REGION Network 54: Reset CMS
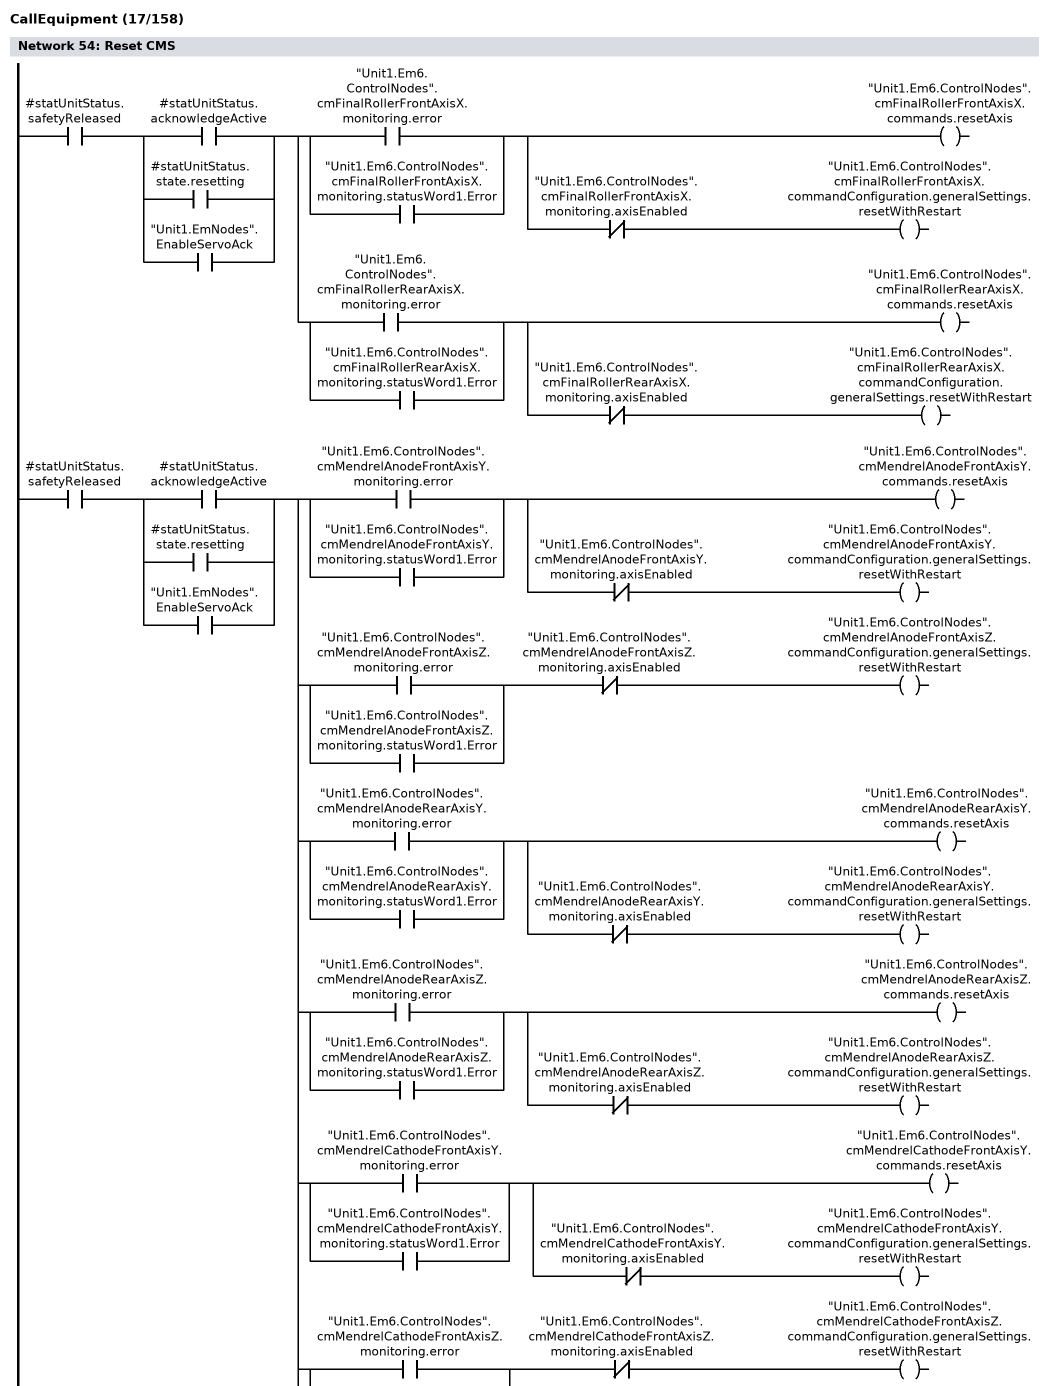
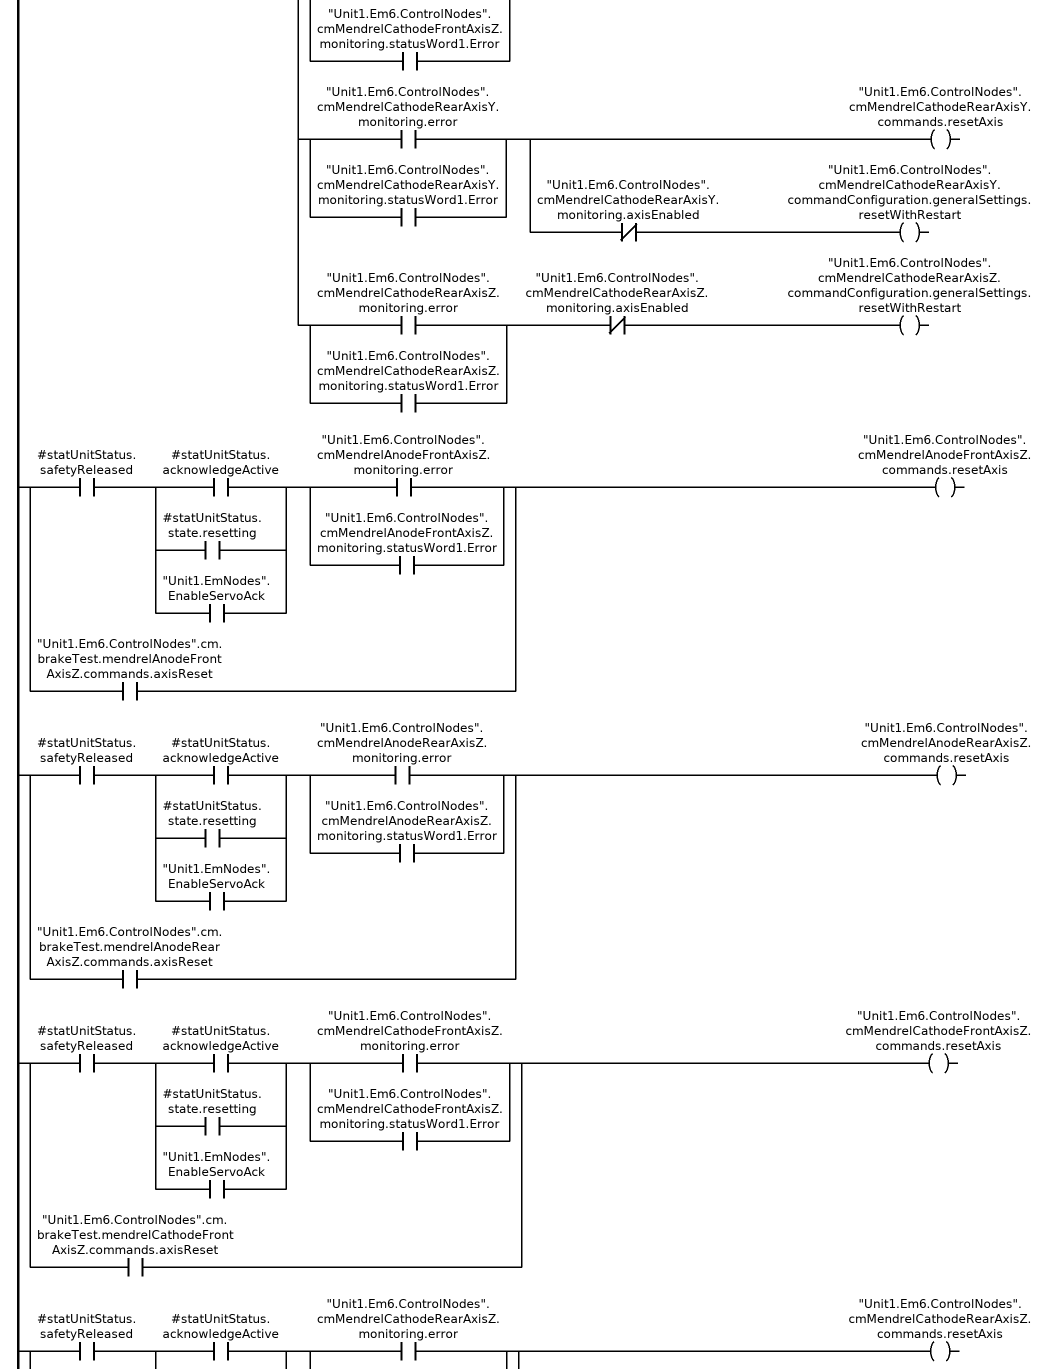
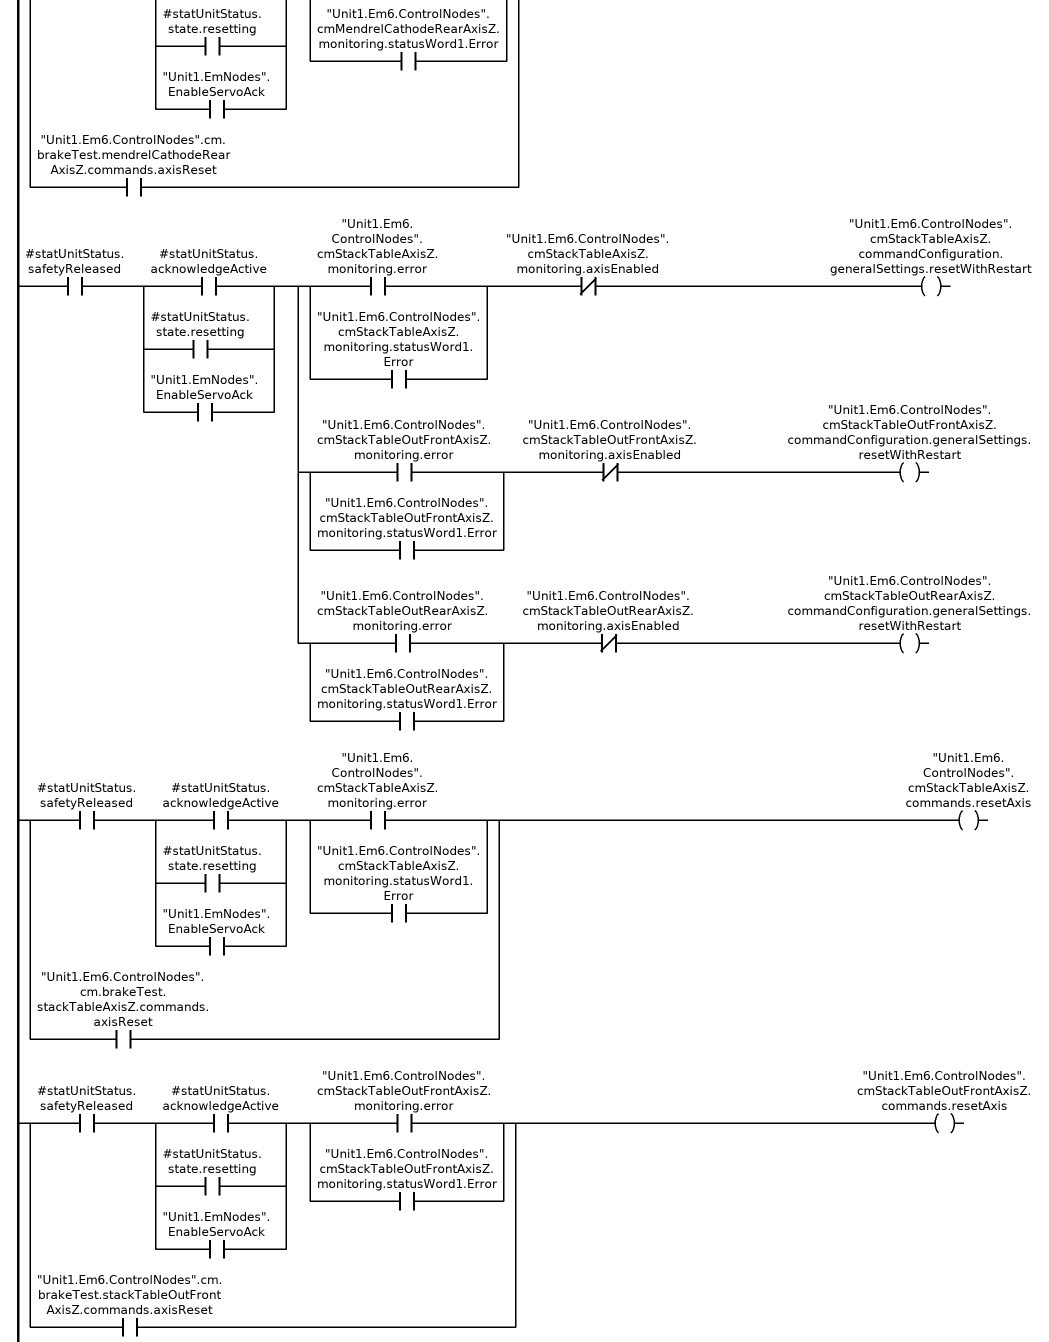
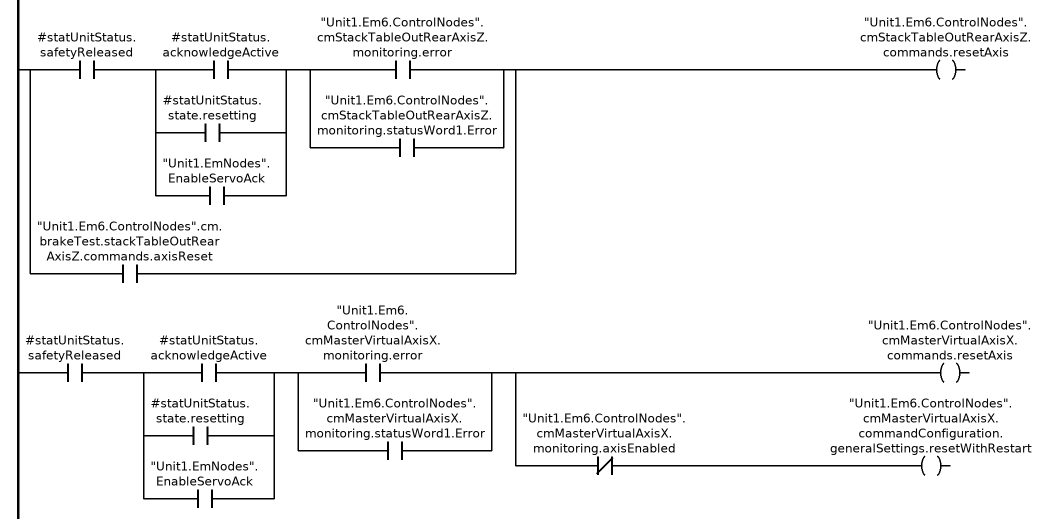
   RUNG wire#powerrail
      Contact( #statUnitStatus.safetyReleased )
      wire#w1
      Contact( #statUnitStatus.acknowledgeActive )
      wire#w2
      Contact( "Unit1.Em6.ControlNodes".cmFinalRollerFrontAxisX.monitoring.error )
      wire#w3
      Coil( "Unit1.Em6.ControlNodes".cmFinalRollerFrontAxisX.commands.resetAxis )
   END_RUNG
   RUNG wire#w1
      Contact( #statUnitStatus.state.resetting )
   END_RUNG wire#w2
   RUNG wire#w1
      Contact( "Unit1.EmNodes".EnableServoAck )
   END_RUNG wire#w2
   RUNG wire#w2
      Contact( "Unit1.Em6.ControlNodes".cmFinalRollerFrontAxisX.monitoring.statusWord1.Error )
   END_RUNG wire#w3
   RUNG wire#w3
      I_Contact( "Unit1.Em6.ControlNodes".cmFinalRollerFrontAxisX.monitoring.axisEnabled )
      Coil( "Unit1.Em6.ControlNodes".cmFinalRollerFrontAxisX.commandConfiguration.generalSettings.resetWithRestart )
   END_RUNG
   RUNG wire#w2
      Contact( "Unit1.Em6.ControlNodes".cmFinalRollerRearAxisX.monitoring.error )
      wire#w4
      Coil( "Unit1.Em6.ControlNodes".cmFinalRollerRearAxisX.commands.resetAxis )
   END_RUNG
   RUNG wire#w2
      Contact( "Unit1.Em6.ControlNodes".cmFinalRollerRearAxisX.monitoring.statusWord1.Error )
   END_RUNG wire#w4
   RUNG wire#w4
      I_Contact( "Unit1.Em6.ControlNodes".cmFinalRollerRearAxisX.monitoring.axisEnabled )
      Coil( "Unit1.Em6.ControlNodes".cmFinalRollerRearAxisX.commandConfiguration.generalSettings.resetWithRestart )
   END_RUNG
   RUNG wire#powerrail
      Contact( #statUnitStatus.safetyReleased )
      wire#w5
      Contact( #statUnitStatus.acknowledgeActive )
      wire#w6
      Contact( "Unit1.Em6.ControlNodes".cmMendrelAnodeFrontAxisY.monitoring.error )
      wire#w7
      Coil( "Unit1.Em6.ControlNodes".cmMendrelAnodeFrontAxisY.commands.resetAxis )
   END_RUNG
   RUNG wire#w5
      Contact( #statUnitStatus.state.resetting )
   END_RUNG wire#w6
   RUNG wire#w5
      Contact( "Unit1.EmNodes".EnableServoAck )
   END_RUNG wire#w6
   RUNG wire#w6
      Contact( "Unit1.Em6.ControlNodes".cmMendrelAnodeFrontAxisY.monitoring.statusWord1.Error )
   END_RUNG wire#w7
   RUNG wire#w7
      I_Contact( "Unit1.Em6.ControlNodes".cmMendrelAnodeFrontAxisY.monitoring.axisEnabled )
      Coil( "Unit1.Em6.ControlNodes".cmMendrelAnodeFrontAxisY.commandConfiguration.generalSettings.resetWithRestart )
   END_RUNG
   RUNG wire#w6
      Contact( "Unit1.Em6.ControlNodes".cmMendrelAnodeFrontAxisZ.monitoring.error )
      wire#w8
      I_Contact( "Unit1.Em6.ControlNodes".cmMendrelAnodeFrontAxisZ.monitoring.axisEnabled )
      Coil( "Unit1.Em6.ControlNodes".cmMendrelAnodeFrontAxisZ.commandConfiguration.generalSettings.resetWithRestart )
   END_RUNG
   RUNG wire#w6
      Contact( "Unit1.Em6.ControlNodes".cmMendrelAnodeFrontAxisZ.monitoring.statusWord1.Error )
   END_RUNG wire#w8
   RUNG wire#w6
      Contact( "Unit1.Em6.ControlNodes".cmMendrelAnodeRearAxisY.monitoring.error )
      wire#w9
      Coil( "Unit1.Em6.ControlNodes".cmMendrelAnodeRearAxisY.commands.resetAxis )
   END_RUNG
   RUNG wire#w6
      Contact( "Unit1.Em6.ControlNodes".cmMendrelAnodeRearAxisY.monitoring.statusWord1.Error )
   END_RUNG wire#w9
   RUNG wire#w9
      I_Contact( "Unit1.Em6.ControlNodes".cmMendrelAnodeRearAxisY.monitoring.axisEnabled )
      Coil( "Unit1.Em6.ControlNodes".cmMendrelAnodeRearAxisY.commandConfiguration.generalSettings.resetWithRestart )
   END_RUNG
   RUNG wire#w6
      Contact( "Unit1.Em6.ControlNodes".cmMendrelAnodeRearAxisZ.monitoring.error )
      wire#w10
      Coil( "Unit1.Em6.ControlNodes".cmMendrelAnodeRearAxisZ.commands.resetAxis )
   END_RUNG
   RUNG wire#w6
      Contact( "Unit1.Em6.ControlNodes".cmMendrelAnodeRearAxisZ.monitoring.statusWord1.Error )
   END_RUNG wire#w10
   RUNG wire#w10
      I_Contact( "Unit1.Em6.ControlNodes".cmMendrelAnodeRearAxisZ.monitoring.axisEnabled )
      Coil( "Unit1.Em6.ControlNodes".cmMendrelAnodeRearAxisZ.commandConfiguration.generalSettings.resetWithRestart )
   END_RUNG
   RUNG wire#w6
      Contact( "Unit1.Em6.ControlNodes".cmMendrelCathodeFrontAxisY.monitoring.error )
      wire#w11
      Coil( "Unit1.Em6.ControlNodes".cmMendrelCathodeFrontAxisY.commands.resetAxis )
   END_RUNG
   RUNG wire#w6
      Contact( "Unit1.Em6.ControlNodes".cmMendrelCathodeFrontAxisY.monitoring.statusWord1.Error )
   END_RUNG wire#w11
   RUNG wire#w11
      I_Contact( "Unit1.Em6.ControlNodes".cmMendrelCathodeFrontAxisY.monitoring.axisEnabled )
      Coil( "Unit1.Em6.ControlNodes".cmMendrelCathodeFrontAxisY.commandConfiguration.generalSettings.resetWithRestart )
   END_RUNG
   RUNG wire#w6
      Contact( "Unit1.Em6.ControlNodes".cmMendrelCathodeFrontAxisZ.monitoring.error )
      wire#w12
      I_Contact( "Unit1.Em6.ControlNodes".cmMendrelCathodeFrontAxisZ.monitoring.axisEnabled )
      Coil( "Unit1.Em6.ControlNodes".cmMendrelCathodeFrontAxisZ.commandConfiguration.generalSettings.resetWithRestart )
   END_RUNG
   RUNG wire#w6
      Contact( "Unit1.Em6.ControlNodes".cmMendrelCathodeFrontAxisZ.monitoring.statusWord1.Error )
   END_RUNG wire#w12
   RUNG wire#w6
      Contact( "Unit1.Em6.ControlNodes".cmMendrelCathodeRearAxisY.monitoring.error )
      wire#w13
      Coil( "Unit1.Em6.ControlNodes".cmMendrelCathodeRearAxisY.commands.resetAxis )
   END_RUNG
   RUNG wire#w6
      Contact( "Unit1.Em6.ControlNodes".cmMendrelCathodeRearAxisY.monitoring.statusWord1.Error )
   END_RUNG wire#w13
   RUNG wire#w13
      I_Contact( "Unit1.Em6.ControlNodes".cmMendrelCathodeRearAxisY.monitoring.axisEnabled )
      Coil( "Unit1.Em6.ControlNodes".cmMendrelCathodeRearAxisY.commandConfiguration.generalSettings.resetWithRestart )
   END_RUNG
   RUNG wire#w6
      Contact( "Unit1.Em6.ControlNodes".cmMendrelCathodeRearAxisZ.monitoring.error )
      wire#w14
      I_Contact( "Unit1.Em6.ControlNodes".cmMendrelCathodeRearAxisZ.monitoring.axisEnabled )
      Coil( "Unit1.Em6.ControlNodes".cmMendrelCathodeRearAxisZ.commandConfiguration.generalSettings.resetWithRestart )
   END_RUNG
   RUNG wire#w6
      Contact( "Unit1.Em6.ControlNodes".cmMendrelCathodeRearAxisZ.monitoring.statusWord1.Error )
   END_RUNG wire#w14
   RUNG wire#powerrail
      Contact( #statUnitStatus.safetyReleased )
      wire#w15
      Contact( #statUnitStatus.acknowledgeActive )
      wire#w16
      Contact( "Unit1.Em6.ControlNodes".cmMendrelAnodeFrontAxisZ.monitoring.error )
      wire#w17
      Coil( "Unit1.Em6.ControlNodes".cmMendrelAnodeFrontAxisZ.commands.resetAxis )
   END_RUNG
   RUNG wire#w15
      Contact( #statUnitStatus.state.resetting )
   END_RUNG wire#w16
   RUNG wire#w15
      Contact( "Unit1.EmNodes".EnableServoAck )
   END_RUNG wire#w16
   RUNG wire#w16
      Contact( "Unit1.Em6.ControlNodes".cmMendrelAnodeFrontAxisZ.monitoring.statusWord1.Error )
   END_RUNG wire#w17
   RUNG wire#powerrail
      Contact( "Unit1.Em6.ControlNodes".cm.brakeTest.mendrelAnodeFrontAxisZ.commands.axisReset )
   END_RUNG wire#w17
   RUNG wire#powerrail
      Contact( #statUnitStatus.safetyReleased )
      wire#w18
      Contact( #statUnitStatus.acknowledgeActive )
      wire#w19
      Contact( "Unit1.Em6.ControlNodes".cmMendrelAnodeRearAxisZ.monitoring.error )
      wire#w20
      Coil( "Unit1.Em6.ControlNodes".cmMendrelAnodeRearAxisZ.commands.resetAxis )
   END_RUNG
   RUNG wire#w18
      Contact( #statUnitStatus.state.resetting )
   END_RUNG wire#w19
   RUNG wire#w18
      Contact( "Unit1.EmNodes".EnableServoAck )
   END_RUNG wire#w19
   RUNG wire#w19
      Contact( "Unit1.Em6.ControlNodes".cmMendrelAnodeRearAxisZ.monitoring.statusWord1.Error )
   END_RUNG wire#w20
   RUNG wire#powerrail
      Contact( "Unit1.Em6.ControlNodes".cm.brakeTest.mendrelAnodeRearAxisZ.commands.axisReset )
   END_RUNG wire#w20
   RUNG wire#powerrail
      Contact( #statUnitStatus.safetyReleased )
      wire#w21
      Contact( #statUnitStatus.acknowledgeActive )
      wire#w22
      Contact( "Unit1.Em6.ControlNodes".cmMendrelCathodeFrontAxisZ.monitoring.error )
      wire#w23
      Coil( "Unit1.Em6.ControlNodes".cmMendrelCathodeFrontAxisZ.commands.resetAxis )
   END_RUNG
   RUNG wire#w21
      Contact( #statUnitStatus.state.resetting )
   END_RUNG wire#w22
   RUNG wire#w21
      Contact( "Unit1.EmNodes".EnableServoAck )
   END_RUNG wire#w22
   RUNG wire#w22
      Contact( "Unit1.Em6.ControlNodes".cmMendrelCathodeFrontAxisZ.monitoring.statusWord1.Error )
   END_RUNG wire#w23
   RUNG wire#powerrail
      Contact( "Unit1.Em6.ControlNodes".cm.brakeTest.mendrelCathodeFrontAxisZ.commands.axisReset )
   END_RUNG wire#w23
   RUNG wire#powerrail
      Contact( #statUnitStatus.safetyReleased )
      wire#w24
      Contact( #statUnitStatus.acknowledgeActive )
      wire#w25
      Contact( "Unit1.Em6.ControlNodes".cmMendrelCathodeRearAxisZ.monitoring.error )
      wire#w26
      Coil( "Unit1.Em6.ControlNodes".cmMendrelCathodeRearAxisZ.commands.resetAxis )
   END_RUNG
   RUNG wire#w24
      Contact( #statUnitStatus.state.resetting )
   END_RUNG wire#w25
   RUNG wire#w24
      Contact( "Unit1.EmNodes".EnableServoAck )
   END_RUNG wire#w25
   RUNG wire#w25
      Contact( "Unit1.Em6.ControlNodes".cmMendrelCathodeRearAxisZ.monitoring.statusWord1.Error )
   END_RUNG wire#w26
   RUNG wire#powerrail
      Contact( "Unit1.Em6.ControlNodes".cm.brakeTest.mendrelCathodeRearAxisZ.commands.axisReset )
   END_RUNG wire#w26
   RUNG wire#powerrail
      Contact( #statUnitStatus.safetyReleased )
      wire#w27
      Contact( #statUnitStatus.acknowledgeActive )
      wire#w28
      Contact( "Unit1.Em6.ControlNodes".cmStackTableAxisZ.monitoring.error )
      wire#w29
      I_Contact( "Unit1.Em6.ControlNodes".cmStackTableAxisZ.monitoring.axisEnabled )
      Coil( "Unit1.Em6.ControlNodes".cmStackTableAxisZ.commandConfiguration.generalSettings.resetWithRestart )
   END_RUNG
   RUNG wire#w27
      Contact( #statUnitStatus.state.resetting )
   END_RUNG wire#w28
   RUNG wire#w27
      Contact( "Unit1.EmNodes".EnableServoAck )
   END_RUNG wire#w28
   RUNG wire#w28
      Contact( "Unit1.Em6.ControlNodes".cmStackTableAxisZ.monitoring.statusWord1.Error )
   END_RUNG wire#w29
   RUNG wire#w28
      Contact( "Unit1.Em6.ControlNodes".cmStackTableOutFrontAxisZ.monitoring.error )
      wire#w30
      I_Contact( "Unit1.Em6.ControlNodes".cmStackTableOutFrontAxisZ.monitoring.axisEnabled )
      Coil( "Unit1.Em6.ControlNodes".cmStackTableOutFrontAxisZ.commandConfiguration.generalSettings.resetWithRestart )
   END_RUNG
   RUNG wire#w28
      Contact( "Unit1.Em6.ControlNodes".cmStackTableOutFrontAxisZ.monitoring.statusWord1.Error )
   END_RUNG wire#w30
   RUNG wire#w28
      Contact( "Unit1.Em6.ControlNodes".cmStackTableOutRearAxisZ.monitoring.error )
      wire#w31
      I_Contact( "Unit1.Em6.ControlNodes".cmStackTableOutRearAxisZ.monitoring.axisEnabled )
      Coil( "Unit1.Em6.ControlNodes".cmStackTableOutRearAxisZ.commandConfiguration.generalSettings.resetWithRestart )
   END_RUNG
   RUNG wire#w28
      Contact( "Unit1.Em6.ControlNodes".cmStackTableOutRearAxisZ.monitoring.statusWord1.Error )
   END_RUNG wire#w31
   RUNG wire#powerrail
      Contact( #statUnitStatus.safetyReleased )
      wire#w32
      Contact( #statUnitStatus.acknowledgeActive )
      wire#w33
      Contact( "Unit1.Em6.ControlNodes".cmStackTableAxisZ.monitoring.error )
      wire#w34
      Coil( "Unit1.Em6.ControlNodes".cmStackTableAxisZ.commands.resetAxis )
   END_RUNG
   RUNG wire#w32
      Contact( #statUnitStatus.state.resetting )
   END_RUNG wire#w33
   RUNG wire#w32
      Contact( "Unit1.EmNodes".EnableServoAck )
   END_RUNG wire#w33
   RUNG wire#w33
      Contact( "Unit1.Em6.ControlNodes".cmStackTableAxisZ.monitoring.statusWord1.Error )
   END_RUNG wire#w34
   RUNG wire#powerrail
      Contact( "Unit1.Em6.ControlNodes".cm.brakeTest.stackTableAxisZ.commands.axisReset )
   END_RUNG wire#w34
   RUNG wire#powerrail
      Contact( #statUnitStatus.safetyReleased )
      wire#w35
      Contact( #statUnitStatus.acknowledgeActive )
      wire#w36
      Contact( "Unit1.Em6.ControlNodes".cmStackTableOutFrontAxisZ.monitoring.error )
      wire#w37
      Coil( "Unit1.Em6.ControlNodes".cmStackTableOutFrontAxisZ.commands.resetAxis )
   END_RUNG
   RUNG wire#w35
      Contact( #statUnitStatus.state.resetting )
   END_RUNG wire#w36
   RUNG wire#w35
      Contact( "Unit1.EmNodes".EnableServoAck )
   END_RUNG wire#w36
   RUNG wire#w36
      Contact( "Unit1.Em6.ControlNodes".cmStackTableOutFrontAxisZ.monitoring.statusWord1.Error )
   END_RUNG wire#w37
   RUNG wire#powerrail
      Contact( "Unit1.Em6.ControlNodes".cm.brakeTest.stackTableOutFrontAxisZ.commands.axisReset )
   END_RUNG wire#w37
   RUNG wire#powerrail
      Contact( #statUnitStatus.safetyReleased )
      wire#w38
      Contact( #statUnitStatus.acknowledgeActive )
      wire#w39
      Contact( "Unit1.Em6.ControlNodes".cmStackTableOutRearAxisZ.monitoring.error )
      wire#w40
      Coil( "Unit1.Em6.ControlNodes".cmStackTableOutRearAxisZ.commands.resetAxis )
   END_RUNG
   RUNG wire#w38
      Contact( #statUnitStatus.state.resetting )
   END_RUNG wire#w39
   RUNG wire#w38
      Contact( "Unit1.EmNodes".EnableServoAck )
   END_RUNG wire#w39
   RUNG wire#w39
      Contact( "Unit1.Em6.ControlNodes".cmStackTableOutRearAxisZ.monitoring.statusWord1.Error )
   END_RUNG wire#w40
   RUNG wire#powerrail
      Contact( "Unit1.Em6.ControlNodes".cm.brakeTest.stackTableOutRearAxisZ.commands.axisReset )
   END_RUNG wire#w40
   RUNG wire#powerrail
      Contact( #statUnitStatus.safetyReleased )
      wire#w41
      Contact( #statUnitStatus.acknowledgeActive )
      wire#w42
      Contact( "Unit1.Em6.ControlNodes".cmMasterVirtualAxisX.monitoring.error )
      wire#w43
      Coil( "Unit1.Em6.ControlNodes".cmMasterVirtualAxisX.commands.resetAxis )
   END_RUNG
   RUNG wire#w41
      Contact( #statUnitStatus.state.resetting )
   END_RUNG wire#w42
   RUNG wire#w41
      Contact( "Unit1.EmNodes".EnableServoAck )
   END_RUNG wire#w42
   RUNG wire#w42
      Contact( "Unit1.Em6.ControlNodes".cmMasterVirtualAxisX.monitoring.statusWord1.Error )
   END_RUNG wire#w43
   RUNG wire#w43
      I_Contact( "Unit1.Em6.ControlNodes".cmMasterVirtualAxisX.monitoring.axisEnabled )
      Coil( "Unit1.Em6.ControlNodes".cmMasterVirtualAxisX.commandConfiguration.generalSettings.resetWithRestart )
   END_RUNG
   // the same network as SCL:
   #_w1 := #statUnitStatus.safetyReleased AND (#statUnitStatus.acknowledgeActive OR #statUnitStatus.state.resetting OR "Unit1.EmNodes".EnableServoAck);
   "Unit1.Em6.ControlNodes".cmFinalRollerFrontAxisX.commands.resetAxis := #_w1 AND ("Unit1.Em6.ControlNodes".cmFinalRollerFrontAxisX.monitoring.error OR "Unit1.Em6.ControlNodes".cmFinalRollerFrontAxisX.monitoring.statusWord1.Error);
   "Unit1.Em6.ControlNodes".cmFinalRollerFrontAxisX.commandConfiguration.generalSettings.resetWithRestart := "Unit1.Em6.ControlNodes".cmFinalRollerFrontAxisX.commands.resetAxis AND NOT "Unit1.Em6.ControlNodes".cmFinalRollerFrontAxisX.monitoring.axisEnabled;
   "Unit1.Em6.ControlNodes".cmFinalRollerRearAxisX.commands.resetAxis := #_w1 AND ("Unit1.Em6.ControlNodes".cmFinalRollerRearAxisX.monitoring.error OR "Unit1.Em6.ControlNodes".cmFinalRollerRearAxisX.monitoring.statusWord1.Error);
   "Unit1.Em6.ControlNodes".cmFinalRollerRearAxisX.commandConfiguration.generalSettings.resetWithRestart := "Unit1.Em6.ControlNodes".cmFinalRollerRearAxisX.commands.resetAxis AND NOT "Unit1.Em6.ControlNodes".cmFinalRollerRearAxisX.monitoring.axisEnabled;
   #_w2 := #statUnitStatus.safetyReleased AND (#statUnitStatus.acknowledgeActive OR #statUnitStatus.state.resetting OR "Unit1.EmNodes".EnableServoAck);
   "Unit1.Em6.ControlNodes".cmMendrelAnodeFrontAxisY.commands.resetAxis := #_w2 AND ("Unit1.Em6.ControlNodes".cmMendrelAnodeFrontAxisY.monitoring.error OR "Unit1.Em6.ControlNodes".cmMendrelAnodeFrontAxisY.monitoring.statusWord1.Error);
   "Unit1.Em6.ControlNodes".cmMendrelAnodeFrontAxisY.commandConfiguration.generalSettings.resetWithRestart := "Unit1.Em6.ControlNodes".cmMendrelAnodeFrontAxisY.commands.resetAxis AND NOT "Unit1.Em6.ControlNodes".cmMendrelAnodeFrontAxisY.monitoring.axisEnabled;
   "Unit1.Em6.ControlNodes".cmMendrelAnodeFrontAxisZ.commandConfiguration.generalSettings.resetWithRestart := #_w2 AND ("Unit1.Em6.ControlNodes".cmMendrelAnodeFrontAxisZ.monitoring.error OR "Unit1.Em6.ControlNodes".cmMendrelAnodeFrontAxisZ.monitoring.statusWord1.Error) AND NOT "Unit1.Em6.ControlNodes".cmMendrelAnodeFrontAxisZ.monitoring.axisEnabled;
   "Unit1.Em6.ControlNodes".cmMendrelAnodeRearAxisY.commands.resetAxis := #_w2 AND ("Unit1.Em6.ControlNodes".cmMendrelAnodeRearAxisY.monitoring.error OR "Unit1.Em6.ControlNodes".cmMendrelAnodeRearAxisY.monitoring.statusWord1.Error);
   "Unit1.Em6.ControlNodes".cmMendrelAnodeRearAxisY.commandConfiguration.generalSettings.resetWithRestart := "Unit1.Em6.ControlNodes".cmMendrelAnodeRearAxisY.commands.resetAxis AND NOT "Unit1.Em6.ControlNodes".cmMendrelAnodeRearAxisY.monitoring.axisEnabled;
   "Unit1.Em6.ControlNodes".cmMendrelAnodeRearAxisZ.commands.resetAxis := #_w2 AND ("Unit1.Em6.ControlNodes".cmMendrelAnodeRearAxisZ.monitoring.error OR "Unit1.Em6.ControlNodes".cmMendrelAnodeRearAxisZ.monitoring.statusWord1.Error);
   "Unit1.Em6.ControlNodes".cmMendrelAnodeRearAxisZ.commandConfiguration.generalSettings.resetWithRestart := "Unit1.Em6.ControlNodes".cmMendrelAnodeRearAxisZ.commands.resetAxis AND NOT "Unit1.Em6.ControlNodes".cmMendrelAnodeRearAxisZ.monitoring.axisEnabled;
   "Unit1.Em6.ControlNodes".cmMendrelCathodeFrontAxisY.commands.resetAxis := #_w2 AND ("Unit1.Em6.ControlNodes".cmMendrelCathodeFrontAxisY.monitoring.error OR "Unit1.Em6.ControlNodes".cmMendrelCathodeFrontAxisY.monitoring.statusWord1.Error);
   "Unit1.Em6.ControlNodes".cmMendrelCathodeFrontAxisY.commandConfiguration.generalSettings.resetWithRestart := "Unit1.Em6.ControlNodes".cmMendrelCathodeFrontAxisY.commands.resetAxis AND NOT "Unit1.Em6.ControlNodes".cmMendrelCathodeFrontAxisY.monitoring.axisEnabled;
   "Unit1.Em6.ControlNodes".cmMendrelCathodeFrontAxisZ.commandConfiguration.generalSettings.resetWithRestart := #_w2 AND ("Unit1.Em6.ControlNodes".cmMendrelCathodeFrontAxisZ.monitoring.error OR "Unit1.Em6.ControlNodes".cmMendrelCathodeFrontAxisZ.monitoring.statusWord1.Error) AND NOT "Unit1.Em6.ControlNodes".cmMendrelCathodeFrontAxisZ.monitoring.axisEnabled;
   "Unit1.Em6.ControlNodes".cmMendrelCathodeRearAxisY.commands.resetAxis := #_w2 AND ("Unit1.Em6.ControlNodes".cmMendrelCathodeRearAxisY.monitoring.error OR "Unit1.Em6.ControlNodes".cmMendrelCathodeRearAxisY.monitoring.statusWord1.Error);
   "Unit1.Em6.ControlNodes".cmMendrelCathodeRearAxisY.commandConfiguration.generalSettings.resetWithRestart := "Unit1.Em6.ControlNodes".cmMendrelCathodeRearAxisY.commands.resetAxis AND NOT "Unit1.Em6.ControlNodes".cmMendrelCathodeRearAxisY.monitoring.axisEnabled;
   "Unit1.Em6.ControlNodes".cmMendrelCathodeRearAxisZ.commandConfiguration.generalSettings.resetWithRestart := #_w2 AND ("Unit1.Em6.ControlNodes".cmMendrelCathodeRearAxisZ.monitoring.error OR "Unit1.Em6.ControlNodes".cmMendrelCathodeRearAxisZ.monitoring.statusWord1.Error) AND NOT "Unit1.Em6.ControlNodes".cmMendrelCathodeRearAxisZ.monitoring.axisEnabled;
   "Unit1.Em6.ControlNodes".cmMendrelAnodeFrontAxisZ.commands.resetAxis := (#statUnitStatus.safetyReleased AND (#statUnitStatus.acknowledgeActive OR #statUnitStatus.state.resetting OR "Unit1.EmNodes".EnableServoAck) AND ("Unit1.Em6.ControlNodes".cmMendrelAnodeFrontAxisZ.monitoring.error OR "Unit1.Em6.ControlNodes".cmMendrelAnodeFrontAxisZ.monitoring.statusWord1.Error)) OR "Unit1.Em6.ControlNodes".cm.brakeTest.mendrelAnodeFrontAxisZ.commands.axisReset;
   "Unit1.Em6.ControlNodes".cmMendrelAnodeRearAxisZ.commands.resetAxis := (#statUnitStatus.safetyReleased AND (#statUnitStatus.acknowledgeActive OR #statUnitStatus.state.resetting OR "Unit1.EmNodes".EnableServoAck) AND ("Unit1.Em6.ControlNodes".cmMendrelAnodeRearAxisZ.monitoring.error OR "Unit1.Em6.ControlNodes".cmMendrelAnodeRearAxisZ.monitoring.statusWord1.Error)) OR "Unit1.Em6.ControlNodes".cm.brakeTest.mendrelAnodeRearAxisZ.commands.axisReset;
   "Unit1.Em6.ControlNodes".cmMendrelCathodeFrontAxisZ.commands.resetAxis := (#statUnitStatus.safetyReleased AND (#statUnitStatus.acknowledgeActive OR #statUnitStatus.state.resetting OR "Unit1.EmNodes".EnableServoAck) AND ("Unit1.Em6.ControlNodes".cmMendrelCathodeFrontAxisZ.monitoring.error OR "Unit1.Em6.ControlNodes".cmMendrelCathodeFrontAxisZ.monitoring.statusWord1.Error)) OR "Unit1.Em6.ControlNodes".cm.brakeTest.mendrelCathodeFrontAxisZ.commands.axisReset;
   "Unit1.Em6.ControlNodes".cmMendrelCathodeRearAxisZ.commands.resetAxis := (#statUnitStatus.safetyReleased AND (#statUnitStatus.acknowledgeActive OR #statUnitStatus.state.resetting OR "Unit1.EmNodes".EnableServoAck) AND ("Unit1.Em6.ControlNodes".cmMendrelCathodeRearAxisZ.monitoring.error OR "Unit1.Em6.ControlNodes".cmMendrelCathodeRearAxisZ.monitoring.statusWord1.Error)) OR "Unit1.Em6.ControlNodes".cm.brakeTest.mendrelCathodeRearAxisZ.commands.axisReset;
   #_w3 := #statUnitStatus.safetyReleased AND (#statUnitStatus.acknowledgeActive OR #statUnitStatus.state.resetting OR "Unit1.EmNodes".EnableServoAck);
   "Unit1.Em6.ControlNodes".cmStackTableAxisZ.commandConfiguration.generalSettings.resetWithRestart := #_w3 AND ("Unit1.Em6.ControlNodes".cmStackTableAxisZ.monitoring.error OR "Unit1.Em6.ControlNodes".cmStackTableAxisZ.monitoring.statusWord1.Error) AND NOT "Unit1.Em6.ControlNodes".cmStackTableAxisZ.monitoring.axisEnabled;
   "Unit1.Em6.ControlNodes".cmStackTableOutFrontAxisZ.commandConfiguration.generalSettings.resetWithRestart := #_w3 AND ("Unit1.Em6.ControlNodes".cmStackTableOutFrontAxisZ.monitoring.error OR "Unit1.Em6.ControlNodes".cmStackTableOutFrontAxisZ.monitoring.statusWord1.Error) AND NOT "Unit1.Em6.ControlNodes".cmStackTableOutFrontAxisZ.monitoring.axisEnabled;
   "Unit1.Em6.ControlNodes".cmStackTableOutRearAxisZ.commandConfiguration.generalSettings.resetWithRestart := #_w3 AND ("Unit1.Em6.ControlNodes".cmStackTableOutRearAxisZ.monitoring.error OR "Unit1.Em6.ControlNodes".cmStackTableOutRearAxisZ.monitoring.statusWord1.Error) AND NOT "Unit1.Em6.ControlNodes".cmStackTableOutRearAxisZ.monitoring.axisEnabled;
   "Unit1.Em6.ControlNodes".cmStackTableAxisZ.commands.resetAxis := (#statUnitStatus.safetyReleased AND (#statUnitStatus.acknowledgeActive OR #statUnitStatus.state.resetting OR "Unit1.EmNodes".EnableServoAck) AND ("Unit1.Em6.ControlNodes".cmStackTableAxisZ.monitoring.error OR "Unit1.Em6.ControlNodes".cmStackTableAxisZ.monitoring.statusWord1.Error)) OR "Unit1.Em6.ControlNodes".cm.brakeTest.stackTableAxisZ.commands.axisReset;
   "Unit1.Em6.ControlNodes".cmStackTableOutFrontAxisZ.commands.resetAxis := (#statUnitStatus.safetyReleased AND (#statUnitStatus.acknowledgeActive OR #statUnitStatus.state.resetting OR "Unit1.EmNodes".EnableServoAck) AND ("Unit1.Em6.ControlNodes".cmStackTableOutFrontAxisZ.monitoring.error OR "Unit1.Em6.ControlNodes".cmStackTableOutFrontAxisZ.monitoring.statusWord1.Error)) OR "Unit1.Em6.ControlNodes".cm.brakeTest.stackTableOutFrontAxisZ.commands.axisReset;
   "Unit1.Em6.ControlNodes".cmStackTableOutRearAxisZ.commands.resetAxis := (#statUnitStatus.safetyReleased AND (#statUnitStatus.acknowledgeActive OR #statUnitStatus.state.resetting OR "Unit1.EmNodes".EnableServoAck) AND ("Unit1.Em6.ControlNodes".cmStackTableOutRearAxisZ.monitoring.error OR "Unit1.Em6.ControlNodes".cmStackTableOutRearAxisZ.monitoring.statusWord1.Error)) OR "Unit1.Em6.ControlNodes".cm.brakeTest.stackTableOutRearAxisZ.commands.axisReset;
   "Unit1.Em6.ControlNodes".cmMasterVirtualAxisX.commands.resetAxis := #statUnitStatus.safetyReleased AND (#statUnitStatus.acknowledgeActive OR #statUnitStatus.state.resetting OR "Unit1.EmNodes".EnableServoAck) AND ("Unit1.Em6.ControlNodes".cmMasterVirtualAxisX.monitoring.error OR "Unit1.Em6.ControlNodes".cmMasterVirtualAxisX.monitoring.statusWord1.Error);
   "Unit1.Em6.ControlNodes".cmMasterVirtualAxisX.commandConfiguration.generalSettings.resetWithRestart := "Unit1.Em6.ControlNodes".cmMasterVirtualAxisX.commands.resetAxis AND NOT "Unit1.Em6.ControlNodes".cmMasterVirtualAxisX.monitoring.axisEnabled;
END_REGION

REGION Network 55: Enable/Disable CMs
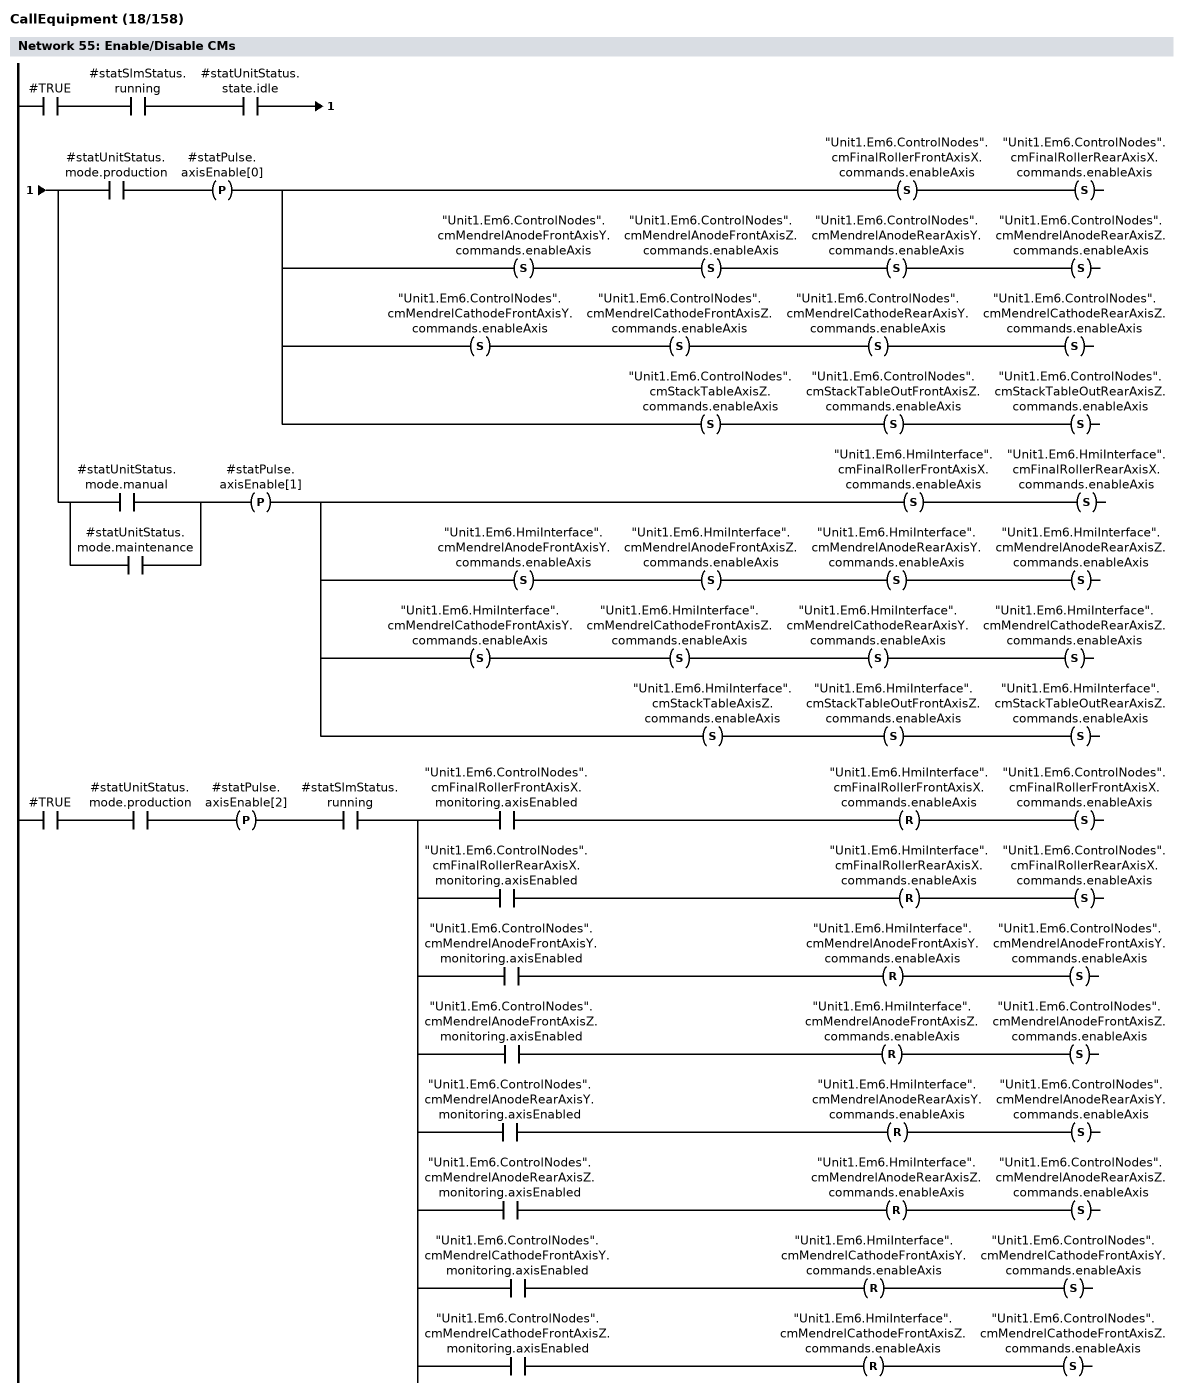
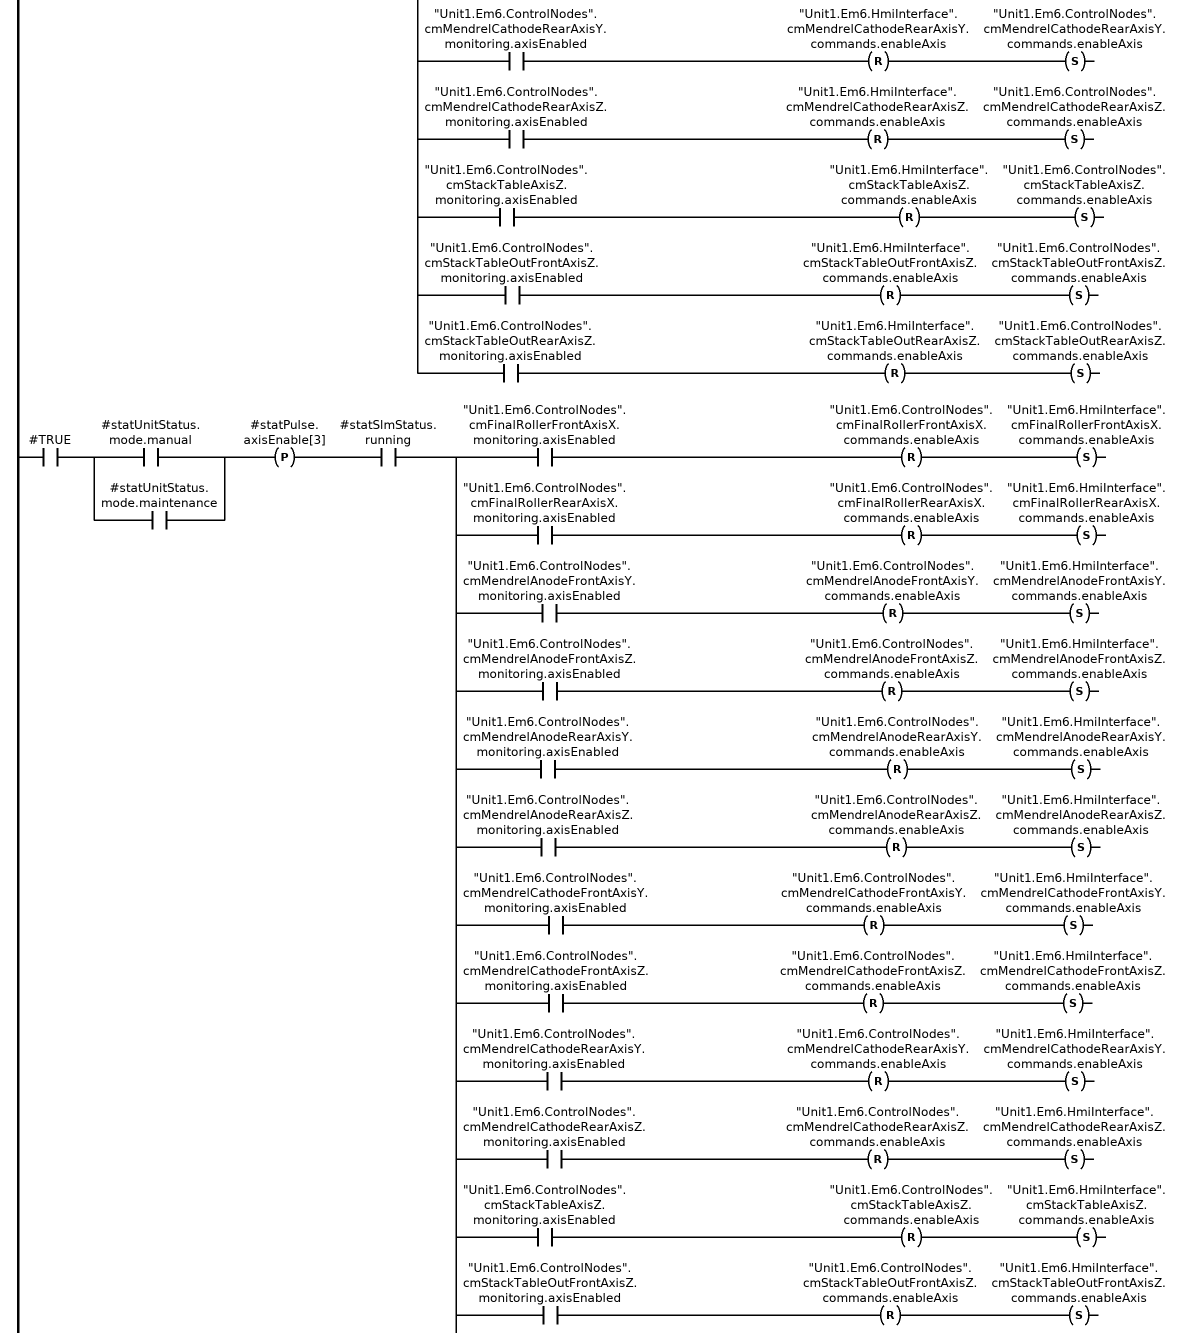
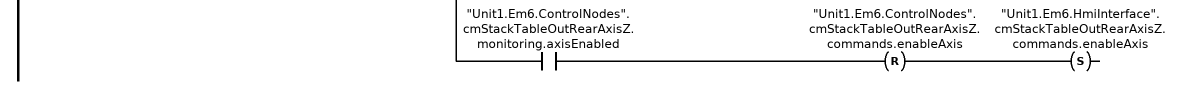
   RUNG wire#powerrail
      Contact( #TRUE )
      Contact( #statSlmStatus.running )
      Contact( #statUnitStatus.state.idle )
      wire#w1
      Contact( #statUnitStatus.mode.production )
      P_Trig( #statPulse.axisEnable[0] )
      wire#w2
      S_Coil( "Unit1.Em6.ControlNodes".cmFinalRollerFrontAxisX.commands.enableAxis )
      S_Coil( "Unit1.Em6.ControlNodes".cmFinalRollerRearAxisX.commands.enableAxis )
   END_RUNG
   RUNG wire#w2
      S_Coil( "Unit1.Em6.ControlNodes".cmMendrelAnodeFrontAxisY.commands.enableAxis )
      S_Coil( "Unit1.Em6.ControlNodes".cmMendrelAnodeFrontAxisZ.commands.enableAxis )
      S_Coil( "Unit1.Em6.ControlNodes".cmMendrelAnodeRearAxisY.commands.enableAxis )
      S_Coil( "Unit1.Em6.ControlNodes".cmMendrelAnodeRearAxisZ.commands.enableAxis )
   END_RUNG
   RUNG wire#w2
      S_Coil( "Unit1.Em6.ControlNodes".cmMendrelCathodeFrontAxisY.commands.enableAxis )
      S_Coil( "Unit1.Em6.ControlNodes".cmMendrelCathodeFrontAxisZ.commands.enableAxis )
      S_Coil( "Unit1.Em6.ControlNodes".cmMendrelCathodeRearAxisY.commands.enableAxis )
      S_Coil( "Unit1.Em6.ControlNodes".cmMendrelCathodeRearAxisZ.commands.enableAxis )
   END_RUNG
   RUNG wire#w2
      S_Coil( "Unit1.Em6.ControlNodes".cmStackTableAxisZ.commands.enableAxis )
      S_Coil( "Unit1.Em6.ControlNodes".cmStackTableOutFrontAxisZ.commands.enableAxis )
      S_Coil( "Unit1.Em6.ControlNodes".cmStackTableOutRearAxisZ.commands.enableAxis )
   END_RUNG
   RUNG wire#w1
      Contact( #statUnitStatus.mode.manual )
      wire#w3
      P_Trig( #statPulse.axisEnable[1] )
      wire#w4
      S_Coil( "Unit1.Em6.HmiInterface".cmFinalRollerFrontAxisX.commands.enableAxis )
      S_Coil( "Unit1.Em6.HmiInterface".cmFinalRollerRearAxisX.commands.enableAxis )
   END_RUNG
   RUNG wire#w1
      Contact( #statUnitStatus.mode.maintenance )
   END_RUNG wire#w3
   RUNG wire#w4
      S_Coil( "Unit1.Em6.HmiInterface".cmMendrelAnodeFrontAxisY.commands.enableAxis )
      S_Coil( "Unit1.Em6.HmiInterface".cmMendrelAnodeFrontAxisZ.commands.enableAxis )
      S_Coil( "Unit1.Em6.HmiInterface".cmMendrelAnodeRearAxisY.commands.enableAxis )
      S_Coil( "Unit1.Em6.HmiInterface".cmMendrelAnodeRearAxisZ.commands.enableAxis )
   END_RUNG
   RUNG wire#w4
      S_Coil( "Unit1.Em6.HmiInterface".cmMendrelCathodeFrontAxisY.commands.enableAxis )
      S_Coil( "Unit1.Em6.HmiInterface".cmMendrelCathodeFrontAxisZ.commands.enableAxis )
      S_Coil( "Unit1.Em6.HmiInterface".cmMendrelCathodeRearAxisY.commands.enableAxis )
      S_Coil( "Unit1.Em6.HmiInterface".cmMendrelCathodeRearAxisZ.commands.enableAxis )
   END_RUNG
   RUNG wire#w4
      S_Coil( "Unit1.Em6.HmiInterface".cmStackTableAxisZ.commands.enableAxis )
      S_Coil( "Unit1.Em6.HmiInterface".cmStackTableOutFrontAxisZ.commands.enableAxis )
      S_Coil( "Unit1.Em6.HmiInterface".cmStackTableOutRearAxisZ.commands.enableAxis )
   END_RUNG
   RUNG wire#powerrail
      Contact( #TRUE )
      Contact( #statUnitStatus.mode.production )
      P_Trig( #statPulse.axisEnable[2] )
      Contact( #statSlmStatus.running )
      wire#w5
      Contact( "Unit1.Em6.ControlNodes".cmFinalRollerFrontAxisX.monitoring.axisEnabled )
      R_Coil( "Unit1.Em6.HmiInterface".cmFinalRollerFrontAxisX.commands.enableAxis )
      S_Coil( "Unit1.Em6.ControlNodes".cmFinalRollerFrontAxisX.commands.enableAxis )
   END_RUNG
   RUNG wire#w5
      Contact( "Unit1.Em6.ControlNodes".cmFinalRollerRearAxisX.monitoring.axisEnabled )
      R_Coil( "Unit1.Em6.HmiInterface".cmFinalRollerRearAxisX.commands.enableAxis )
      S_Coil( "Unit1.Em6.ControlNodes".cmFinalRollerRearAxisX.commands.enableAxis )
   END_RUNG
   RUNG wire#w5
      Contact( "Unit1.Em6.ControlNodes".cmMendrelAnodeFrontAxisY.monitoring.axisEnabled )
      R_Coil( "Unit1.Em6.HmiInterface".cmMendrelAnodeFrontAxisY.commands.enableAxis )
      S_Coil( "Unit1.Em6.ControlNodes".cmMendrelAnodeFrontAxisY.commands.enableAxis )
   END_RUNG
   RUNG wire#w5
      Contact( "Unit1.Em6.ControlNodes".cmMendrelAnodeFrontAxisZ.monitoring.axisEnabled )
      R_Coil( "Unit1.Em6.HmiInterface".cmMendrelAnodeFrontAxisZ.commands.enableAxis )
      S_Coil( "Unit1.Em6.ControlNodes".cmMendrelAnodeFrontAxisZ.commands.enableAxis )
   END_RUNG
   RUNG wire#w5
      Contact( "Unit1.Em6.ControlNodes".cmMendrelAnodeRearAxisY.monitoring.axisEnabled )
      R_Coil( "Unit1.Em6.HmiInterface".cmMendrelAnodeRearAxisY.commands.enableAxis )
      S_Coil( "Unit1.Em6.ControlNodes".cmMendrelAnodeRearAxisY.commands.enableAxis )
   END_RUNG
   RUNG wire#w5
      Contact( "Unit1.Em6.ControlNodes".cmMendrelAnodeRearAxisZ.monitoring.axisEnabled )
      R_Coil( "Unit1.Em6.HmiInterface".cmMendrelAnodeRearAxisZ.commands.enableAxis )
      S_Coil( "Unit1.Em6.ControlNodes".cmMendrelAnodeRearAxisZ.commands.enableAxis )
   END_RUNG
   RUNG wire#w5
      Contact( "Unit1.Em6.ControlNodes".cmMendrelCathodeFrontAxisY.monitoring.axisEnabled )
      R_Coil( "Unit1.Em6.HmiInterface".cmMendrelCathodeFrontAxisY.commands.enableAxis )
      S_Coil( "Unit1.Em6.ControlNodes".cmMendrelCathodeFrontAxisY.commands.enableAxis )
   END_RUNG
   RUNG wire#w5
      Contact( "Unit1.Em6.ControlNodes".cmMendrelCathodeFrontAxisZ.monitoring.axisEnabled )
      R_Coil( "Unit1.Em6.HmiInterface".cmMendrelCathodeFrontAxisZ.commands.enableAxis )
      S_Coil( "Unit1.Em6.ControlNodes".cmMendrelCathodeFrontAxisZ.commands.enableAxis )
   END_RUNG
   RUNG wire#w5
      Contact( "Unit1.Em6.ControlNodes".cmMendrelCathodeRearAxisY.monitoring.axisEnabled )
      R_Coil( "Unit1.Em6.HmiInterface".cmMendrelCathodeRearAxisY.commands.enableAxis )
      S_Coil( "Unit1.Em6.ControlNodes".cmMendrelCathodeRearAxisY.commands.enableAxis )
   END_RUNG
   RUNG wire#w5
      Contact( "Unit1.Em6.ControlNodes".cmMendrelCathodeRearAxisZ.monitoring.axisEnabled )
      R_Coil( "Unit1.Em6.HmiInterface".cmMendrelCathodeRearAxisZ.commands.enableAxis )
      S_Coil( "Unit1.Em6.ControlNodes".cmMendrelCathodeRearAxisZ.commands.enableAxis )
   END_RUNG
   RUNG wire#w5
      Contact( "Unit1.Em6.ControlNodes".cmStackTableAxisZ.monitoring.axisEnabled )
      R_Coil( "Unit1.Em6.HmiInterface".cmStackTableAxisZ.commands.enableAxis )
      S_Coil( "Unit1.Em6.ControlNodes".cmStackTableAxisZ.commands.enableAxis )
   END_RUNG
   RUNG wire#w5
      Contact( "Unit1.Em6.ControlNodes".cmStackTableOutFrontAxisZ.monitoring.axisEnabled )
      R_Coil( "Unit1.Em6.HmiInterface".cmStackTableOutFrontAxisZ.commands.enableAxis )
      S_Coil( "Unit1.Em6.ControlNodes".cmStackTableOutFrontAxisZ.commands.enableAxis )
   END_RUNG
   RUNG wire#w5
      Contact( "Unit1.Em6.ControlNodes".cmStackTableOutRearAxisZ.monitoring.axisEnabled )
      R_Coil( "Unit1.Em6.HmiInterface".cmStackTableOutRearAxisZ.commands.enableAxis )
      S_Coil( "Unit1.Em6.ControlNodes".cmStackTableOutRearAxisZ.commands.enableAxis )
   END_RUNG
   RUNG wire#powerrail
      Contact( #TRUE )
      wire#w6
      Contact( #statUnitStatus.mode.manual )
      wire#w7
      P_Trig( #statPulse.axisEnable[3] )
      Contact( #statSlmStatus.running )
      wire#w8
      Contact( "Unit1.Em6.ControlNodes".cmFinalRollerFrontAxisX.monitoring.axisEnabled )
      R_Coil( "Unit1.Em6.ControlNodes".cmFinalRollerFrontAxisX.commands.enableAxis )
      S_Coil( "Unit1.Em6.HmiInterface".cmFinalRollerFrontAxisX.commands.enableAxis )
   END_RUNG
   RUNG wire#w6
      Contact( #statUnitStatus.mode.maintenance )
   END_RUNG wire#w7
   RUNG wire#w8
      Contact( "Unit1.Em6.ControlNodes".cmFinalRollerRearAxisX.monitoring.axisEnabled )
      R_Coil( "Unit1.Em6.ControlNodes".cmFinalRollerRearAxisX.commands.enableAxis )
      S_Coil( "Unit1.Em6.HmiInterface".cmFinalRollerRearAxisX.commands.enableAxis )
   END_RUNG
   RUNG wire#w8
      Contact( "Unit1.Em6.ControlNodes".cmMendrelAnodeFrontAxisY.monitoring.axisEnabled )
      R_Coil( "Unit1.Em6.ControlNodes".cmMendrelAnodeFrontAxisY.commands.enableAxis )
      S_Coil( "Unit1.Em6.HmiInterface".cmMendrelAnodeFrontAxisY.commands.enableAxis )
   END_RUNG
   RUNG wire#w8
      Contact( "Unit1.Em6.ControlNodes".cmMendrelAnodeFrontAxisZ.monitoring.axisEnabled )
      R_Coil( "Unit1.Em6.ControlNodes".cmMendrelAnodeFrontAxisZ.commands.enableAxis )
      S_Coil( "Unit1.Em6.HmiInterface".cmMendrelAnodeFrontAxisZ.commands.enableAxis )
   END_RUNG
   RUNG wire#w8
      Contact( "Unit1.Em6.ControlNodes".cmMendrelAnodeRearAxisY.monitoring.axisEnabled )
      R_Coil( "Unit1.Em6.ControlNodes".cmMendrelAnodeRearAxisY.commands.enableAxis )
      S_Coil( "Unit1.Em6.HmiInterface".cmMendrelAnodeRearAxisY.commands.enableAxis )
   END_RUNG
   RUNG wire#w8
      Contact( "Unit1.Em6.ControlNodes".cmMendrelAnodeRearAxisZ.monitoring.axisEnabled )
      R_Coil( "Unit1.Em6.ControlNodes".cmMendrelAnodeRearAxisZ.commands.enableAxis )
      S_Coil( "Unit1.Em6.HmiInterface".cmMendrelAnodeRearAxisZ.commands.enableAxis )
   END_RUNG
   RUNG wire#w8
      Contact( "Unit1.Em6.ControlNodes".cmMendrelCathodeFrontAxisY.monitoring.axisEnabled )
      R_Coil( "Unit1.Em6.ControlNodes".cmMendrelCathodeFrontAxisY.commands.enableAxis )
      S_Coil( "Unit1.Em6.HmiInterface".cmMendrelCathodeFrontAxisY.commands.enableAxis )
   END_RUNG
   RUNG wire#w8
      Contact( "Unit1.Em6.ControlNodes".cmMendrelCathodeFrontAxisZ.monitoring.axisEnabled )
      R_Coil( "Unit1.Em6.ControlNodes".cmMendrelCathodeFrontAxisZ.commands.enableAxis )
      S_Coil( "Unit1.Em6.HmiInterface".cmMendrelCathodeFrontAxisZ.commands.enableAxis )
   END_RUNG
   RUNG wire#w8
      Contact( "Unit1.Em6.ControlNodes".cmMendrelCathodeRearAxisY.monitoring.axisEnabled )
      R_Coil( "Unit1.Em6.ControlNodes".cmMendrelCathodeRearAxisY.commands.enableAxis )
      S_Coil( "Unit1.Em6.HmiInterface".cmMendrelCathodeRearAxisY.commands.enableAxis )
   END_RUNG
   RUNG wire#w8
      Contact( "Unit1.Em6.ControlNodes".cmMendrelCathodeRearAxisZ.monitoring.axisEnabled )
      R_Coil( "Unit1.Em6.ControlNodes".cmMendrelCathodeRearAxisZ.commands.enableAxis )
      S_Coil( "Unit1.Em6.HmiInterface".cmMendrelCathodeRearAxisZ.commands.enableAxis )
   END_RUNG
   RUNG wire#w8
      Contact( "Unit1.Em6.ControlNodes".cmStackTableAxisZ.monitoring.axisEnabled )
      R_Coil( "Unit1.Em6.ControlNodes".cmStackTableAxisZ.commands.enableAxis )
      S_Coil( "Unit1.Em6.HmiInterface".cmStackTableAxisZ.commands.enableAxis )
   END_RUNG
   RUNG wire#w8
      Contact( "Unit1.Em6.ControlNodes".cmStackTableOutFrontAxisZ.monitoring.axisEnabled )
      R_Coil( "Unit1.Em6.ControlNodes".cmStackTableOutFrontAxisZ.commands.enableAxis )
      S_Coil( "Unit1.Em6.HmiInterface".cmStackTableOutFrontAxisZ.commands.enableAxis )
   END_RUNG
   RUNG wire#w8
      Contact( "Unit1.Em6.ControlNodes".cmStackTableOutRearAxisZ.monitoring.axisEnabled )
      R_Coil( "Unit1.Em6.ControlNodes".cmStackTableOutRearAxisZ.commands.enableAxis )
      S_Coil( "Unit1.Em6.HmiInterface".cmStackTableOutRearAxisZ.commands.enableAxis )
   END_RUNG
   // the same network as SCL:
   #_w1 := #TRUE AND #statSlmStatus.running AND #statUnitStatus.state.idle;
   #_w2 := #_w1 AND #statUnitStatus.mode.production;
   #_w3 := #_w2 AND NOT #statPulse.axisEnable[0];   // rising edge
   #statPulse.axisEnable[0] := #_w2;
   IF #_w3 THEN
       "Unit1.Em6.ControlNodes".cmFinalRollerFrontAxisX.commands.enableAxis := TRUE;
       "Unit1.Em6.ControlNodes".cmFinalRollerRearAxisX.commands.enableAxis := TRUE;
       "Unit1.Em6.ControlNodes".cmMendrelAnodeFrontAxisY.commands.enableAxis := TRUE;
       "Unit1.Em6.ControlNodes".cmMendrelAnodeFrontAxisZ.commands.enableAxis := TRUE;
       "Unit1.Em6.ControlNodes".cmMendrelAnodeRearAxisY.commands.enableAxis := TRUE;
       "Unit1.Em6.ControlNodes".cmMendrelAnodeRearAxisZ.commands.enableAxis := TRUE;
       "Unit1.Em6.ControlNodes".cmMendrelCathodeFrontAxisY.commands.enableAxis := TRUE;
       "Unit1.Em6.ControlNodes".cmMendrelCathodeFrontAxisZ.commands.enableAxis := TRUE;
       "Unit1.Em6.ControlNodes".cmMendrelCathodeRearAxisY.commands.enableAxis := TRUE;
       "Unit1.Em6.ControlNodes".cmMendrelCathodeRearAxisZ.commands.enableAxis := TRUE;
       "Unit1.Em6.ControlNodes".cmStackTableAxisZ.commands.enableAxis := TRUE;
       "Unit1.Em6.ControlNodes".cmStackTableOutFrontAxisZ.commands.enableAxis := TRUE;
       "Unit1.Em6.ControlNodes".cmStackTableOutRearAxisZ.commands.enableAxis := TRUE;
   END_IF;
   #_w4 := #_w1 AND (#statUnitStatus.mode.manual OR #statUnitStatus.mode.maintenance);
   #_w5 := #_w4 AND NOT #statPulse.axisEnable[1];   // rising edge
   #statPulse.axisEnable[1] := #_w4;
   IF #_w5 THEN
       "Unit1.Em6.HmiInterface".cmFinalRollerFrontAxisX.commands.enableAxis := TRUE;
       "Unit1.Em6.HmiInterface".cmFinalRollerRearAxisX.commands.enableAxis := TRUE;
       "Unit1.Em6.HmiInterface".cmMendrelAnodeFrontAxisY.commands.enableAxis := TRUE;
       "Unit1.Em6.HmiInterface".cmMendrelAnodeFrontAxisZ.commands.enableAxis := TRUE;
       "Unit1.Em6.HmiInterface".cmMendrelAnodeRearAxisY.commands.enableAxis := TRUE;
       "Unit1.Em6.HmiInterface".cmMendrelAnodeRearAxisZ.commands.enableAxis := TRUE;
       "Unit1.Em6.HmiInterface".cmMendrelCathodeFrontAxisY.commands.enableAxis := TRUE;
       "Unit1.Em6.HmiInterface".cmMendrelCathodeFrontAxisZ.commands.enableAxis := TRUE;
       "Unit1.Em6.HmiInterface".cmMendrelCathodeRearAxisY.commands.enableAxis := TRUE;
       "Unit1.Em6.HmiInterface".cmMendrelCathodeRearAxisZ.commands.enableAxis := TRUE;
       "Unit1.Em6.HmiInterface".cmStackTableAxisZ.commands.enableAxis := TRUE;
       "Unit1.Em6.HmiInterface".cmStackTableOutFrontAxisZ.commands.enableAxis := TRUE;
       "Unit1.Em6.HmiInterface".cmStackTableOutRearAxisZ.commands.enableAxis := TRUE;
   END_IF;
   #_w6 := #TRUE AND #statUnitStatus.mode.production;
   #_w7 := #_w6 AND NOT #statPulse.axisEnable[2];   // rising edge
   #statPulse.axisEnable[2] := #_w6;
   #_w8 := #_w7 AND #statSlmStatus.running;
   IF #_w8 AND "Unit1.Em6.ControlNodes".cmFinalRollerFrontAxisX.monitoring.axisEnabled THEN
       "Unit1.Em6.HmiInterface".cmFinalRollerFrontAxisX.commands.enableAxis := FALSE;
       "Unit1.Em6.ControlNodes".cmFinalRollerFrontAxisX.commands.enableAxis := TRUE;
   END_IF;
   IF #_w8 AND "Unit1.Em6.ControlNodes".cmFinalRollerRearAxisX.monitoring.axisEnabled THEN
       "Unit1.Em6.HmiInterface".cmFinalRollerRearAxisX.commands.enableAxis := FALSE;
       "Unit1.Em6.ControlNodes".cmFinalRollerRearAxisX.commands.enableAxis := TRUE;
   END_IF;
   IF #_w8 AND "Unit1.Em6.ControlNodes".cmMendrelAnodeFrontAxisY.monitoring.axisEnabled THEN
       "Unit1.Em6.HmiInterface".cmMendrelAnodeFrontAxisY.commands.enableAxis := FALSE;
       "Unit1.Em6.ControlNodes".cmMendrelAnodeFrontAxisY.commands.enableAxis := TRUE;
   END_IF;
   IF #_w8 AND "Unit1.Em6.ControlNodes".cmMendrelAnodeFrontAxisZ.monitoring.axisEnabled THEN
       "Unit1.Em6.HmiInterface".cmMendrelAnodeFrontAxisZ.commands.enableAxis := FALSE;
       "Unit1.Em6.ControlNodes".cmMendrelAnodeFrontAxisZ.commands.enableAxis := TRUE;
   END_IF;
   IF #_w8 AND "Unit1.Em6.ControlNodes".cmMendrelAnodeRearAxisY.monitoring.axisEnabled THEN
       "Unit1.Em6.HmiInterface".cmMendrelAnodeRearAxisY.commands.enableAxis := FALSE;
       "Unit1.Em6.ControlNodes".cmMendrelAnodeRearAxisY.commands.enableAxis := TRUE;
   END_IF;
   IF #_w8 AND "Unit1.Em6.ControlNodes".cmMendrelAnodeRearAxisZ.monitoring.axisEnabled THEN
       "Unit1.Em6.HmiInterface".cmMendrelAnodeRearAxisZ.commands.enableAxis := FALSE;
       "Unit1.Em6.ControlNodes".cmMendrelAnodeRearAxisZ.commands.enableAxis := TRUE;
   END_IF;
   IF #_w8 AND "Unit1.Em6.ControlNodes".cmMendrelCathodeFrontAxisY.monitoring.axisEnabled THEN
       "Unit1.Em6.HmiInterface".cmMendrelCathodeFrontAxisY.commands.enableAxis := FALSE;
       "Unit1.Em6.ControlNodes".cmMendrelCathodeFrontAxisY.commands.enableAxis := TRUE;
   END_IF;
   IF #_w8 AND "Unit1.Em6.ControlNodes".cmMendrelCathodeFrontAxisZ.monitoring.axisEnabled THEN
       "Unit1.Em6.HmiInterface".cmMendrelCathodeFrontAxisZ.commands.enableAxis := FALSE;
       "Unit1.Em6.ControlNodes".cmMendrelCathodeFrontAxisZ.commands.enableAxis := TRUE;
   END_IF;
   IF #_w8 AND "Unit1.Em6.ControlNodes".cmMendrelCathodeRearAxisY.monitoring.axisEnabled THEN
       "Unit1.Em6.HmiInterface".cmMendrelCathodeRearAxisY.commands.enableAxis := FALSE;
       "Unit1.Em6.ControlNodes".cmMendrelCathodeRearAxisY.commands.enableAxis := TRUE;
   END_IF;
   IF #_w8 AND "Unit1.Em6.ControlNodes".cmMendrelCathodeRearAxisZ.monitoring.axisEnabled THEN
       "Unit1.Em6.HmiInterface".cmMendrelCathodeRearAxisZ.commands.enableAxis := FALSE;
       "Unit1.Em6.ControlNodes".cmMendrelCathodeRearAxisZ.commands.enableAxis := TRUE;
   END_IF;
   IF #_w8 AND "Unit1.Em6.ControlNodes".cmStackTableAxisZ.monitoring.axisEnabled THEN
       "Unit1.Em6.HmiInterface".cmStackTableAxisZ.commands.enableAxis := FALSE;
       "Unit1.Em6.ControlNodes".cmStackTableAxisZ.commands.enableAxis := TRUE;
   END_IF;
   IF #_w8 AND "Unit1.Em6.ControlNodes".cmStackTableOutFrontAxisZ.monitoring.axisEnabled THEN
       "Unit1.Em6.HmiInterface".cmStackTableOutFrontAxisZ.commands.enableAxis := FALSE;
       "Unit1.Em6.ControlNodes".cmStackTableOutFrontAxisZ.commands.enableAxis := TRUE;
   END_IF;
   IF #_w8 AND "Unit1.Em6.ControlNodes".cmStackTableOutRearAxisZ.monitoring.axisEnabled THEN
       "Unit1.Em6.HmiInterface".cmStackTableOutRearAxisZ.commands.enableAxis := FALSE;
       "Unit1.Em6.ControlNodes".cmStackTableOutRearAxisZ.commands.enableAxis := TRUE;
   END_IF;
   #_w9 := #TRUE AND (#statUnitStatus.mode.manual OR #statUnitStatus.mode.maintenance);
   #_w10 := #_w9 AND NOT #statPulse.axisEnable[3];   // rising edge
   #statPulse.axisEnable[3] := #_w9;
   #_w11 := #_w10 AND #statSlmStatus.running;
   IF #_w11 AND "Unit1.Em6.ControlNodes".cmFinalRollerFrontAxisX.monitoring.axisEnabled THEN
       "Unit1.Em6.ControlNodes".cmFinalRollerFrontAxisX.commands.enableAxis := FALSE;
       "Unit1.Em6.HmiInterface".cmFinalRollerFrontAxisX.commands.enableAxis := TRUE;
   END_IF;
   IF #_w11 AND "Unit1.Em6.ControlNodes".cmFinalRollerRearAxisX.monitoring.axisEnabled THEN
       "Unit1.Em6.ControlNodes".cmFinalRollerRearAxisX.commands.enableAxis := FALSE;
       "Unit1.Em6.HmiInterface".cmFinalRollerRearAxisX.commands.enableAxis := TRUE;
   END_IF;
   IF #_w11 AND "Unit1.Em6.ControlNodes".cmMendrelAnodeFrontAxisY.monitoring.axisEnabled THEN
       "Unit1.Em6.ControlNodes".cmMendrelAnodeFrontAxisY.commands.enableAxis := FALSE;
       "Unit1.Em6.HmiInterface".cmMendrelAnodeFrontAxisY.commands.enableAxis := TRUE;
   END_IF;
   IF #_w11 AND "Unit1.Em6.ControlNodes".cmMendrelAnodeFrontAxisZ.monitoring.axisEnabled THEN
       "Unit1.Em6.ControlNodes".cmMendrelAnodeFrontAxisZ.commands.enableAxis := FALSE;
       "Unit1.Em6.HmiInterface".cmMendrelAnodeFrontAxisZ.commands.enableAxis := TRUE;
   END_IF;
   IF #_w11 AND "Unit1.Em6.ControlNodes".cmMendrelAnodeRearAxisY.monitoring.axisEnabled THEN
       "Unit1.Em6.ControlNodes".cmMendrelAnodeRearAxisY.commands.enableAxis := FALSE;
       "Unit1.Em6.HmiInterface".cmMendrelAnodeRearAxisY.commands.enableAxis := TRUE;
   END_IF;
   IF #_w11 AND "Unit1.Em6.ControlNodes".cmMendrelAnodeRearAxisZ.monitoring.axisEnabled THEN
       "Unit1.Em6.ControlNodes".cmMendrelAnodeRearAxisZ.commands.enableAxis := FALSE;
       "Unit1.Em6.HmiInterface".cmMendrelAnodeRearAxisZ.commands.enableAxis := TRUE;
   END_IF;
   IF #_w11 AND "Unit1.Em6.ControlNodes".cmMendrelCathodeFrontAxisY.monitoring.axisEnabled THEN
       "Unit1.Em6.ControlNodes".cmMendrelCathodeFrontAxisY.commands.enableAxis := FALSE;
       "Unit1.Em6.HmiInterface".cmMendrelCathodeFrontAxisY.commands.enableAxis := TRUE;
   END_IF;
   IF #_w11 AND "Unit1.Em6.ControlNodes".cmMendrelCathodeFrontAxisZ.monitoring.axisEnabled THEN
       "Unit1.Em6.ControlNodes".cmMendrelCathodeFrontAxisZ.commands.enableAxis := FALSE;
       "Unit1.Em6.HmiInterface".cmMendrelCathodeFrontAxisZ.commands.enableAxis := TRUE;
   END_IF;
   IF #_w11 AND "Unit1.Em6.ControlNodes".cmMendrelCathodeRearAxisY.monitoring.axisEnabled THEN
       "Unit1.Em6.ControlNodes".cmMendrelCathodeRearAxisY.commands.enableAxis := FALSE;
       "Unit1.Em6.HmiInterface".cmMendrelCathodeRearAxisY.commands.enableAxis := TRUE;
   END_IF;
   IF #_w11 AND "Unit1.Em6.ControlNodes".cmMendrelCathodeRearAxisZ.monitoring.axisEnabled THEN
       "Unit1.Em6.ControlNodes".cmMendrelCathodeRearAxisZ.commands.enableAxis := FALSE;
       "Unit1.Em6.HmiInterface".cmMendrelCathodeRearAxisZ.commands.enableAxis := TRUE;
   END_IF;
   IF #_w11 AND "Unit1.Em6.ControlNodes".cmStackTableAxisZ.monitoring.axisEnabled THEN
       "Unit1.Em6.ControlNodes".cmStackTableAxisZ.commands.enableAxis := FALSE;
       "Unit1.Em6.HmiInterface".cmStackTableAxisZ.commands.enableAxis := TRUE;
   END_IF;
   IF #_w11 AND "Unit1.Em6.ControlNodes".cmStackTableOutFrontAxisZ.monitoring.axisEnabled THEN
       "Unit1.Em6.ControlNodes".cmStackTableOutFrontAxisZ.commands.enableAxis := FALSE;
       "Unit1.Em6.HmiInterface".cmStackTableOutFrontAxisZ.commands.enableAxis := TRUE;
   END_IF;
   IF #_w11 AND "Unit1.Em6.ControlNodes".cmStackTableOutRearAxisZ.monitoring.axisEnabled THEN
       "Unit1.Em6.ControlNodes".cmStackTableOutRearAxisZ.commands.enableAxis := FALSE;
       "Unit1.Em6.HmiInterface".cmStackTableOutRearAxisZ.commands.enableAxis := TRUE;
   END_IF;
END_REGION

REGION Network 56: PHMI Servo Enable CMs
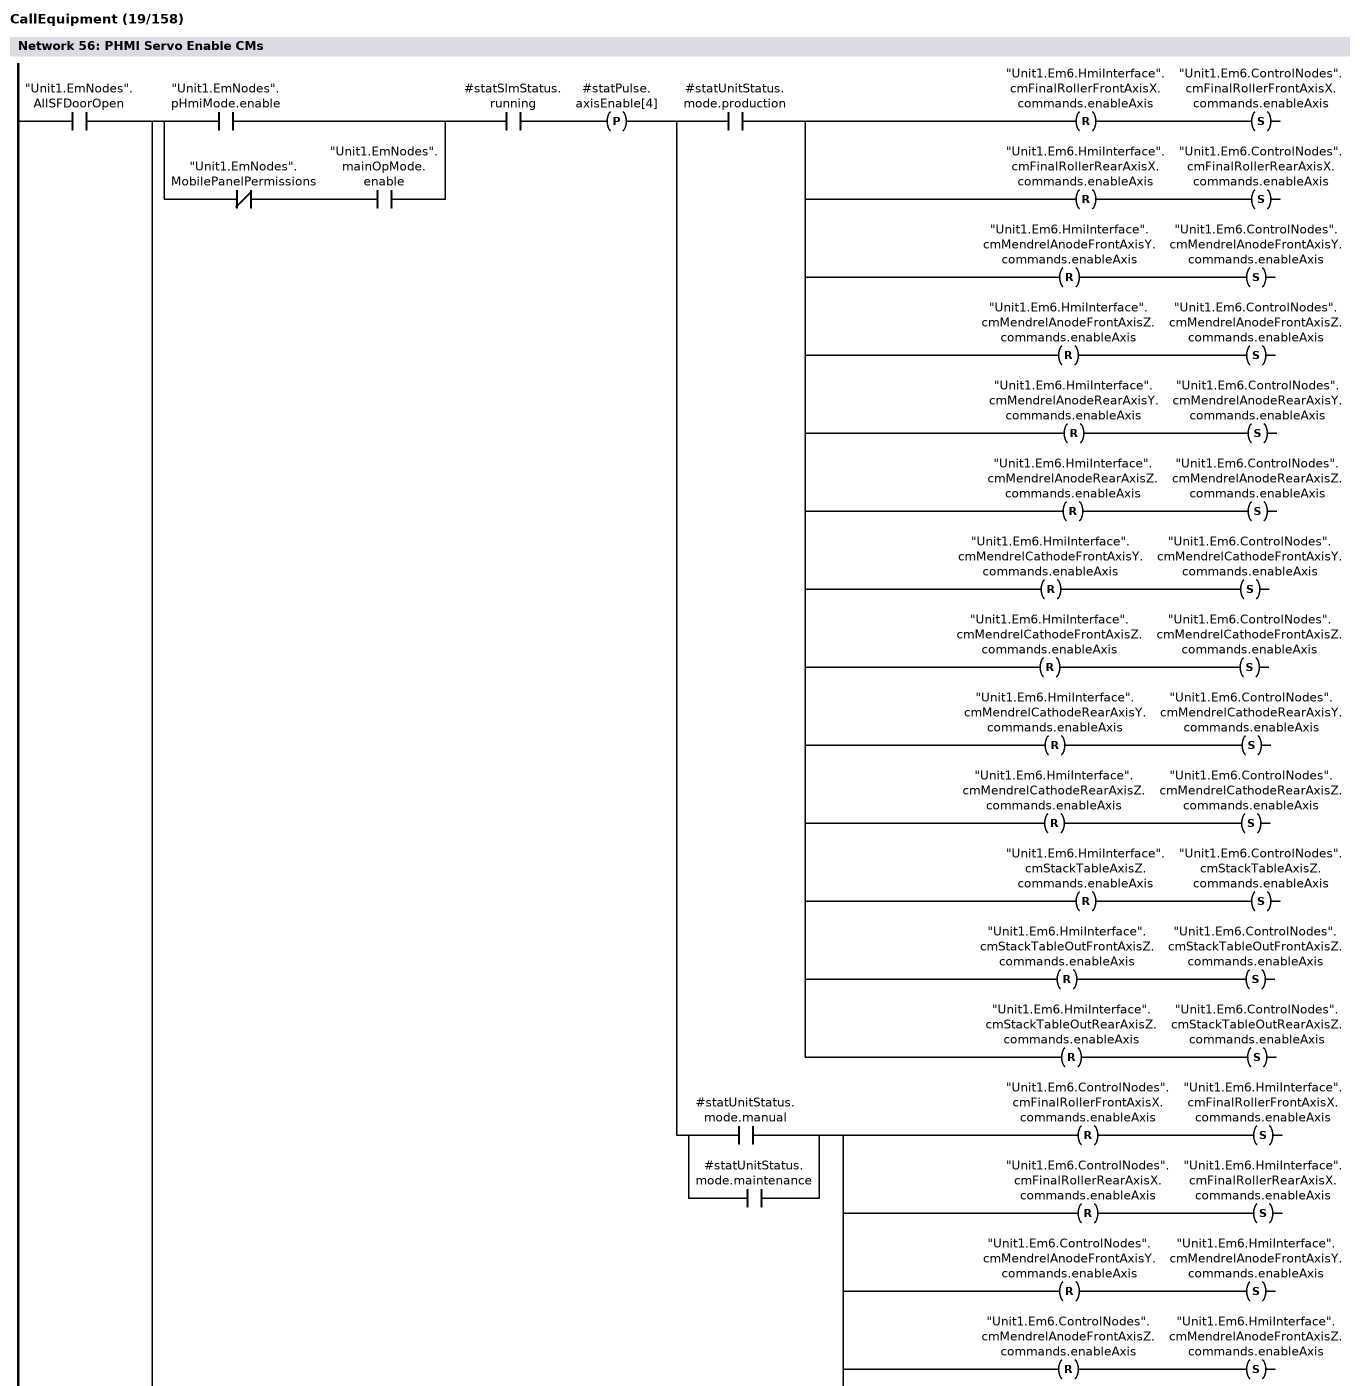
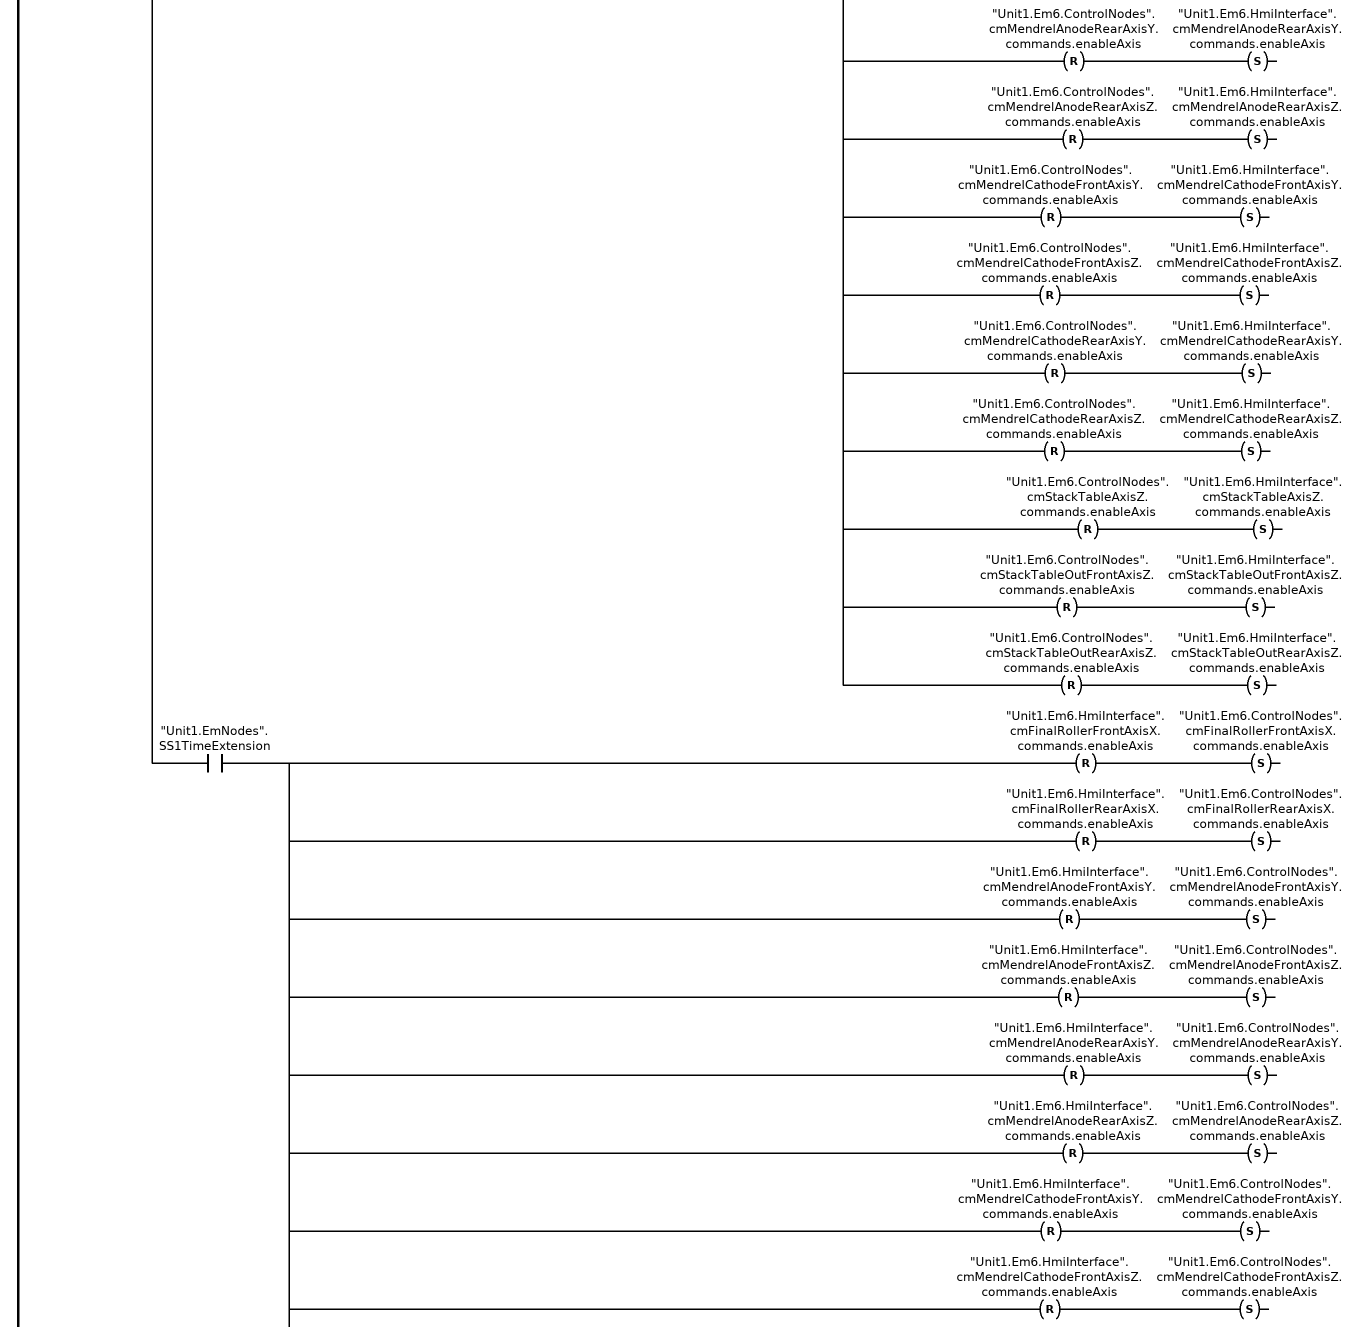
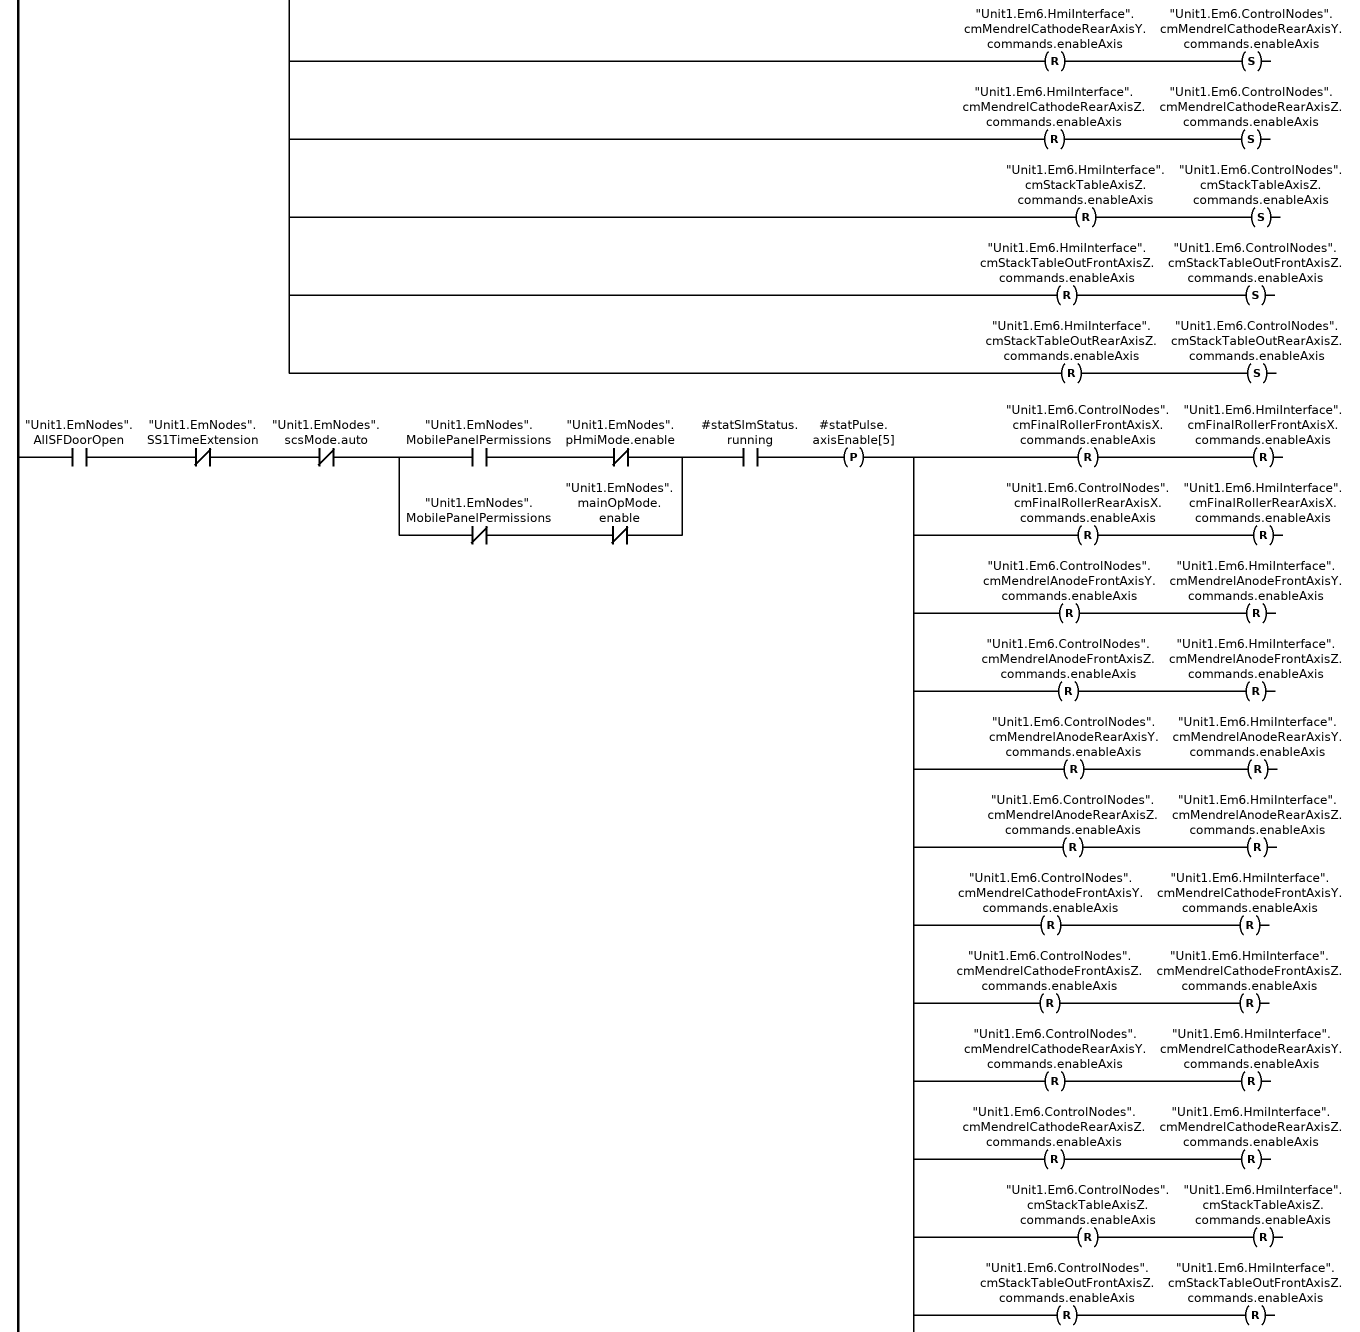
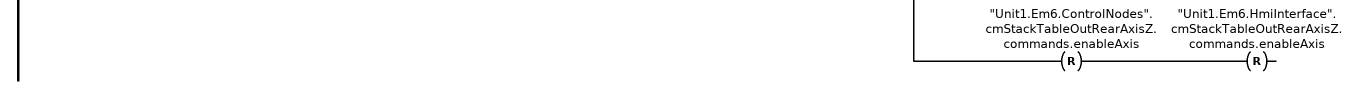
   RUNG wire#powerrail
      Contact( "Unit1.EmNodes".AllSFDoorOpen )
      wire#w1
      Contact( "Unit1.EmNodes".pHmiMode.enable )
      wire#w2
      Contact( #statSlmStatus.running )
      P_Trig( #statPulse.axisEnable[4] )
      wire#w3
      Contact( #statUnitStatus.mode.production )
      wire#w4
      R_Coil( "Unit1.Em6.HmiInterface".cmFinalRollerFrontAxisX.commands.enableAxis )
      S_Coil( "Unit1.Em6.ControlNodes".cmFinalRollerFrontAxisX.commands.enableAxis )
   END_RUNG
   RUNG wire#w1
      I_Contact( "Unit1.EmNodes".MobilePanelPermissions )
      Contact( "Unit1.EmNodes".mainOpMode.enable )
   END_RUNG wire#w2
   RUNG wire#w4
      R_Coil( "Unit1.Em6.HmiInterface".cmFinalRollerRearAxisX.commands.enableAxis )
      S_Coil( "Unit1.Em6.ControlNodes".cmFinalRollerRearAxisX.commands.enableAxis )
   END_RUNG
   RUNG wire#w4
      R_Coil( "Unit1.Em6.HmiInterface".cmMendrelAnodeFrontAxisY.commands.enableAxis )
      S_Coil( "Unit1.Em6.ControlNodes".cmMendrelAnodeFrontAxisY.commands.enableAxis )
   END_RUNG
   RUNG wire#w4
      R_Coil( "Unit1.Em6.HmiInterface".cmMendrelAnodeFrontAxisZ.commands.enableAxis )
      S_Coil( "Unit1.Em6.ControlNodes".cmMendrelAnodeFrontAxisZ.commands.enableAxis )
   END_RUNG
   RUNG wire#w4
      R_Coil( "Unit1.Em6.HmiInterface".cmMendrelAnodeRearAxisY.commands.enableAxis )
      S_Coil( "Unit1.Em6.ControlNodes".cmMendrelAnodeRearAxisY.commands.enableAxis )
   END_RUNG
   RUNG wire#w4
      R_Coil( "Unit1.Em6.HmiInterface".cmMendrelAnodeRearAxisZ.commands.enableAxis )
      S_Coil( "Unit1.Em6.ControlNodes".cmMendrelAnodeRearAxisZ.commands.enableAxis )
   END_RUNG
   RUNG wire#w4
      R_Coil( "Unit1.Em6.HmiInterface".cmMendrelCathodeFrontAxisY.commands.enableAxis )
      S_Coil( "Unit1.Em6.ControlNodes".cmMendrelCathodeFrontAxisY.commands.enableAxis )
   END_RUNG
   RUNG wire#w4
      R_Coil( "Unit1.Em6.HmiInterface".cmMendrelCathodeFrontAxisZ.commands.enableAxis )
      S_Coil( "Unit1.Em6.ControlNodes".cmMendrelCathodeFrontAxisZ.commands.enableAxis )
   END_RUNG
   RUNG wire#w4
      R_Coil( "Unit1.Em6.HmiInterface".cmMendrelCathodeRearAxisY.commands.enableAxis )
      S_Coil( "Unit1.Em6.ControlNodes".cmMendrelCathodeRearAxisY.commands.enableAxis )
   END_RUNG
   RUNG wire#w4
      R_Coil( "Unit1.Em6.HmiInterface".cmMendrelCathodeRearAxisZ.commands.enableAxis )
      S_Coil( "Unit1.Em6.ControlNodes".cmMendrelCathodeRearAxisZ.commands.enableAxis )
   END_RUNG
   RUNG wire#w4
      R_Coil( "Unit1.Em6.HmiInterface".cmStackTableAxisZ.commands.enableAxis )
      S_Coil( "Unit1.Em6.ControlNodes".cmStackTableAxisZ.commands.enableAxis )
   END_RUNG
   RUNG wire#w4
      R_Coil( "Unit1.Em6.HmiInterface".cmStackTableOutFrontAxisZ.commands.enableAxis )
      S_Coil( "Unit1.Em6.ControlNodes".cmStackTableOutFrontAxisZ.commands.enableAxis )
   END_RUNG
   RUNG wire#w4
      R_Coil( "Unit1.Em6.HmiInterface".cmStackTableOutRearAxisZ.commands.enableAxis )
      S_Coil( "Unit1.Em6.ControlNodes".cmStackTableOutRearAxisZ.commands.enableAxis )
   END_RUNG
   RUNG wire#w3
      Contact( #statUnitStatus.mode.manual )
      wire#w5
      R_Coil( "Unit1.Em6.ControlNodes".cmFinalRollerFrontAxisX.commands.enableAxis )
      S_Coil( "Unit1.Em6.HmiInterface".cmFinalRollerFrontAxisX.commands.enableAxis )
   END_RUNG
   RUNG wire#w3
      Contact( #statUnitStatus.mode.maintenance )
   END_RUNG wire#w5
   RUNG wire#w5
      R_Coil( "Unit1.Em6.ControlNodes".cmFinalRollerRearAxisX.commands.enableAxis )
      S_Coil( "Unit1.Em6.HmiInterface".cmFinalRollerRearAxisX.commands.enableAxis )
   END_RUNG
   RUNG wire#w5
      R_Coil( "Unit1.Em6.ControlNodes".cmMendrelAnodeFrontAxisY.commands.enableAxis )
      S_Coil( "Unit1.Em6.HmiInterface".cmMendrelAnodeFrontAxisY.commands.enableAxis )
   END_RUNG
   RUNG wire#w5
      R_Coil( "Unit1.Em6.ControlNodes".cmMendrelAnodeFrontAxisZ.commands.enableAxis )
      S_Coil( "Unit1.Em6.HmiInterface".cmMendrelAnodeFrontAxisZ.commands.enableAxis )
   END_RUNG
   RUNG wire#w5
      R_Coil( "Unit1.Em6.ControlNodes".cmMendrelAnodeRearAxisY.commands.enableAxis )
      S_Coil( "Unit1.Em6.HmiInterface".cmMendrelAnodeRearAxisY.commands.enableAxis )
   END_RUNG
   RUNG wire#w5
      R_Coil( "Unit1.Em6.ControlNodes".cmMendrelAnodeRearAxisZ.commands.enableAxis )
      S_Coil( "Unit1.Em6.HmiInterface".cmMendrelAnodeRearAxisZ.commands.enableAxis )
   END_RUNG
   RUNG wire#w5
      R_Coil( "Unit1.Em6.ControlNodes".cmMendrelCathodeFrontAxisY.commands.enableAxis )
      S_Coil( "Unit1.Em6.HmiInterface".cmMendrelCathodeFrontAxisY.commands.enableAxis )
   END_RUNG
   RUNG wire#w5
      R_Coil( "Unit1.Em6.ControlNodes".cmMendrelCathodeFrontAxisZ.commands.enableAxis )
      S_Coil( "Unit1.Em6.HmiInterface".cmMendrelCathodeFrontAxisZ.commands.enableAxis )
   END_RUNG
   RUNG wire#w5
      R_Coil( "Unit1.Em6.ControlNodes".cmMendrelCathodeRearAxisY.commands.enableAxis )
      S_Coil( "Unit1.Em6.HmiInterface".cmMendrelCathodeRearAxisY.commands.enableAxis )
   END_RUNG
   RUNG wire#w5
      R_Coil( "Unit1.Em6.ControlNodes".cmMendrelCathodeRearAxisZ.commands.enableAxis )
      S_Coil( "Unit1.Em6.HmiInterface".cmMendrelCathodeRearAxisZ.commands.enableAxis )
   END_RUNG
   RUNG wire#w5
      R_Coil( "Unit1.Em6.ControlNodes".cmStackTableAxisZ.commands.enableAxis )
      S_Coil( "Unit1.Em6.HmiInterface".cmStackTableAxisZ.commands.enableAxis )
   END_RUNG
   RUNG wire#w5
      R_Coil( "Unit1.Em6.ControlNodes".cmStackTableOutFrontAxisZ.commands.enableAxis )
      S_Coil( "Unit1.Em6.HmiInterface".cmStackTableOutFrontAxisZ.commands.enableAxis )
   END_RUNG
   RUNG wire#w5
      R_Coil( "Unit1.Em6.ControlNodes".cmStackTableOutRearAxisZ.commands.enableAxis )
      S_Coil( "Unit1.Em6.HmiInterface".cmStackTableOutRearAxisZ.commands.enableAxis )
   END_RUNG
   RUNG wire#w1
      Contact( "Unit1.EmNodes".SS1TimeExtension )
      wire#w6
      R_Coil( "Unit1.Em6.HmiInterface".cmFinalRollerFrontAxisX.commands.enableAxis )
      S_Coil( "Unit1.Em6.ControlNodes".cmFinalRollerFrontAxisX.commands.enableAxis )
   END_RUNG
   RUNG wire#w6
      R_Coil( "Unit1.Em6.HmiInterface".cmFinalRollerRearAxisX.commands.enableAxis )
      S_Coil( "Unit1.Em6.ControlNodes".cmFinalRollerRearAxisX.commands.enableAxis )
   END_RUNG
   RUNG wire#w6
      R_Coil( "Unit1.Em6.HmiInterface".cmMendrelAnodeFrontAxisY.commands.enableAxis )
      S_Coil( "Unit1.Em6.ControlNodes".cmMendrelAnodeFrontAxisY.commands.enableAxis )
   END_RUNG
   RUNG wire#w6
      R_Coil( "Unit1.Em6.HmiInterface".cmMendrelAnodeFrontAxisZ.commands.enableAxis )
      S_Coil( "Unit1.Em6.ControlNodes".cmMendrelAnodeFrontAxisZ.commands.enableAxis )
   END_RUNG
   RUNG wire#w6
      R_Coil( "Unit1.Em6.HmiInterface".cmMendrelAnodeRearAxisY.commands.enableAxis )
      S_Coil( "Unit1.Em6.ControlNodes".cmMendrelAnodeRearAxisY.commands.enableAxis )
   END_RUNG
   RUNG wire#w6
      R_Coil( "Unit1.Em6.HmiInterface".cmMendrelAnodeRearAxisZ.commands.enableAxis )
      S_Coil( "Unit1.Em6.ControlNodes".cmMendrelAnodeRearAxisZ.commands.enableAxis )
   END_RUNG
   RUNG wire#w6
      R_Coil( "Unit1.Em6.HmiInterface".cmMendrelCathodeFrontAxisY.commands.enableAxis )
      S_Coil( "Unit1.Em6.ControlNodes".cmMendrelCathodeFrontAxisY.commands.enableAxis )
   END_RUNG
   RUNG wire#w6
      R_Coil( "Unit1.Em6.HmiInterface".cmMendrelCathodeFrontAxisZ.commands.enableAxis )
      S_Coil( "Unit1.Em6.ControlNodes".cmMendrelCathodeFrontAxisZ.commands.enableAxis )
   END_RUNG
   RUNG wire#w6
      R_Coil( "Unit1.Em6.HmiInterface".cmMendrelCathodeRearAxisY.commands.enableAxis )
      S_Coil( "Unit1.Em6.ControlNodes".cmMendrelCathodeRearAxisY.commands.enableAxis )
   END_RUNG
   RUNG wire#w6
      R_Coil( "Unit1.Em6.HmiInterface".cmMendrelCathodeRearAxisZ.commands.enableAxis )
      S_Coil( "Unit1.Em6.ControlNodes".cmMendrelCathodeRearAxisZ.commands.enableAxis )
   END_RUNG
   RUNG wire#w6
      R_Coil( "Unit1.Em6.HmiInterface".cmStackTableAxisZ.commands.enableAxis )
      S_Coil( "Unit1.Em6.ControlNodes".cmStackTableAxisZ.commands.enableAxis )
   END_RUNG
   RUNG wire#w6
      R_Coil( "Unit1.Em6.HmiInterface".cmStackTableOutFrontAxisZ.commands.enableAxis )
      S_Coil( "Unit1.Em6.ControlNodes".cmStackTableOutFrontAxisZ.commands.enableAxis )
   END_RUNG
   RUNG wire#w6
      R_Coil( "Unit1.Em6.HmiInterface".cmStackTableOutRearAxisZ.commands.enableAxis )
      S_Coil( "Unit1.Em6.ControlNodes".cmStackTableOutRearAxisZ.commands.enableAxis )
   END_RUNG
   RUNG wire#powerrail
      Contact( "Unit1.EmNodes".AllSFDoorOpen )
      I_Contact( "Unit1.EmNodes".SS1TimeExtension )
      I_Contact( "Unit1.EmNodes".scsMode.auto )
      wire#w7
      Contact( "Unit1.EmNodes".MobilePanelPermissions )
      I_Contact( "Unit1.EmNodes".pHmiMode.enable )
      wire#w8
      Contact( #statSlmStatus.running )
      P_Trig( #statPulse.axisEnable[5] )
      wire#w9
      R_Coil( "Unit1.Em6.ControlNodes".cmFinalRollerFrontAxisX.commands.enableAxis )
      R_Coil( "Unit1.Em6.HmiInterface".cmFinalRollerFrontAxisX.commands.enableAxis )
   END_RUNG
   RUNG wire#w7
      I_Contact( "Unit1.EmNodes".MobilePanelPermissions )
      I_Contact( "Unit1.EmNodes".mainOpMode.enable )
   END_RUNG wire#w8
   RUNG wire#w9
      R_Coil( "Unit1.Em6.ControlNodes".cmFinalRollerRearAxisX.commands.enableAxis )
      R_Coil( "Unit1.Em6.HmiInterface".cmFinalRollerRearAxisX.commands.enableAxis )
   END_RUNG
   RUNG wire#w9
      R_Coil( "Unit1.Em6.ControlNodes".cmMendrelAnodeFrontAxisY.commands.enableAxis )
      R_Coil( "Unit1.Em6.HmiInterface".cmMendrelAnodeFrontAxisY.commands.enableAxis )
   END_RUNG
   RUNG wire#w9
      R_Coil( "Unit1.Em6.ControlNodes".cmMendrelAnodeFrontAxisZ.commands.enableAxis )
      R_Coil( "Unit1.Em6.HmiInterface".cmMendrelAnodeFrontAxisZ.commands.enableAxis )
   END_RUNG
   RUNG wire#w9
      R_Coil( "Unit1.Em6.ControlNodes".cmMendrelAnodeRearAxisY.commands.enableAxis )
      R_Coil( "Unit1.Em6.HmiInterface".cmMendrelAnodeRearAxisY.commands.enableAxis )
   END_RUNG
   RUNG wire#w9
      R_Coil( "Unit1.Em6.ControlNodes".cmMendrelAnodeRearAxisZ.commands.enableAxis )
      R_Coil( "Unit1.Em6.HmiInterface".cmMendrelAnodeRearAxisZ.commands.enableAxis )
   END_RUNG
   RUNG wire#w9
      R_Coil( "Unit1.Em6.ControlNodes".cmMendrelCathodeFrontAxisY.commands.enableAxis )
      R_Coil( "Unit1.Em6.HmiInterface".cmMendrelCathodeFrontAxisY.commands.enableAxis )
   END_RUNG
   RUNG wire#w9
      R_Coil( "Unit1.Em6.ControlNodes".cmMendrelCathodeFrontAxisZ.commands.enableAxis )
      R_Coil( "Unit1.Em6.HmiInterface".cmMendrelCathodeFrontAxisZ.commands.enableAxis )
   END_RUNG
   RUNG wire#w9
      R_Coil( "Unit1.Em6.ControlNodes".cmMendrelCathodeRearAxisY.commands.enableAxis )
      R_Coil( "Unit1.Em6.HmiInterface".cmMendrelCathodeRearAxisY.commands.enableAxis )
   END_RUNG
   RUNG wire#w9
      R_Coil( "Unit1.Em6.ControlNodes".cmMendrelCathodeRearAxisZ.commands.enableAxis )
      R_Coil( "Unit1.Em6.HmiInterface".cmMendrelCathodeRearAxisZ.commands.enableAxis )
   END_RUNG
   RUNG wire#w9
      R_Coil( "Unit1.Em6.ControlNodes".cmStackTableAxisZ.commands.enableAxis )
      R_Coil( "Unit1.Em6.HmiInterface".cmStackTableAxisZ.commands.enableAxis )
   END_RUNG
   RUNG wire#w9
      R_Coil( "Unit1.Em6.ControlNodes".cmStackTableOutFrontAxisZ.commands.enableAxis )
      R_Coil( "Unit1.Em6.HmiInterface".cmStackTableOutFrontAxisZ.commands.enableAxis )
   END_RUNG
   RUNG wire#w9
      R_Coil( "Unit1.Em6.ControlNodes".cmStackTableOutRearAxisZ.commands.enableAxis )
      R_Coil( "Unit1.Em6.HmiInterface".cmStackTableOutRearAxisZ.commands.enableAxis )
   END_RUNG
   // the same network as SCL:
   #_w1 := "Unit1.EmNodes".AllSFDoorOpen AND ("Unit1.EmNodes".pHmiMode.enable OR (NOT "Unit1.EmNodes".MobilePanelPermissions AND "Unit1.EmNodes".mainOpMode.enable)) AND #statSlmStatus.running;
   #_w2 := #_w1 AND NOT #statPulse.axisEnable[4];   // rising edge
   #statPulse.axisEnable[4] := #_w1;
   IF #_w2 AND #statUnitStatus.mode.production THEN
       "Unit1.Em6.HmiInterface".cmFinalRollerFrontAxisX.commands.enableAxis := FALSE;
       "Unit1.Em6.ControlNodes".cmFinalRollerFrontAxisX.commands.enableAxis := TRUE;
       "Unit1.Em6.HmiInterface".cmFinalRollerRearAxisX.commands.enableAxis := FALSE;
       "Unit1.Em6.ControlNodes".cmFinalRollerRearAxisX.commands.enableAxis := TRUE;
       "Unit1.Em6.HmiInterface".cmMendrelAnodeFrontAxisY.commands.enableAxis := FALSE;
       "Unit1.Em6.ControlNodes".cmMendrelAnodeFrontAxisY.commands.enableAxis := TRUE;
       "Unit1.Em6.HmiInterface".cmMendrelAnodeFrontAxisZ.commands.enableAxis := FALSE;
       "Unit1.Em6.ControlNodes".cmMendrelAnodeFrontAxisZ.commands.enableAxis := TRUE;
       "Unit1.Em6.HmiInterface".cmMendrelAnodeRearAxisY.commands.enableAxis := FALSE;
       "Unit1.Em6.ControlNodes".cmMendrelAnodeRearAxisY.commands.enableAxis := TRUE;
       "Unit1.Em6.HmiInterface".cmMendrelAnodeRearAxisZ.commands.enableAxis := FALSE;
       "Unit1.Em6.ControlNodes".cmMendrelAnodeRearAxisZ.commands.enableAxis := TRUE;
       "Unit1.Em6.HmiInterface".cmMendrelCathodeFrontAxisY.commands.enableAxis := FALSE;
       "Unit1.Em6.ControlNodes".cmMendrelCathodeFrontAxisY.commands.enableAxis := TRUE;
       "Unit1.Em6.HmiInterface".cmMendrelCathodeFrontAxisZ.commands.enableAxis := FALSE;
       "Unit1.Em6.ControlNodes".cmMendrelCathodeFrontAxisZ.commands.enableAxis := TRUE;
       "Unit1.Em6.HmiInterface".cmMendrelCathodeRearAxisY.commands.enableAxis := FALSE;
       "Unit1.Em6.ControlNodes".cmMendrelCathodeRearAxisY.commands.enableAxis := TRUE;
       "Unit1.Em6.HmiInterface".cmMendrelCathodeRearAxisZ.commands.enableAxis := FALSE;
       "Unit1.Em6.ControlNodes".cmMendrelCathodeRearAxisZ.commands.enableAxis := TRUE;
       "Unit1.Em6.HmiInterface".cmStackTableAxisZ.commands.enableAxis := FALSE;
       "Unit1.Em6.ControlNodes".cmStackTableAxisZ.commands.enableAxis := TRUE;
       "Unit1.Em6.HmiInterface".cmStackTableOutFrontAxisZ.commands.enableAxis := FALSE;
       "Unit1.Em6.ControlNodes".cmStackTableOutFrontAxisZ.commands.enableAxis := TRUE;
       "Unit1.Em6.HmiInterface".cmStackTableOutRearAxisZ.commands.enableAxis := FALSE;
       "Unit1.Em6.ControlNodes".cmStackTableOutRearAxisZ.commands.enableAxis := TRUE;
   END_IF;
   IF #_w2 AND (#statUnitStatus.mode.manual OR #statUnitStatus.mode.maintenance) THEN
       "Unit1.Em6.ControlNodes".cmFinalRollerFrontAxisX.commands.enableAxis := FALSE;
       "Unit1.Em6.HmiInterface".cmFinalRollerFrontAxisX.commands.enableAxis := TRUE;
       "Unit1.Em6.ControlNodes".cmFinalRollerRearAxisX.commands.enableAxis := FALSE;
       "Unit1.Em6.HmiInterface".cmFinalRollerRearAxisX.commands.enableAxis := TRUE;
       "Unit1.Em6.ControlNodes".cmMendrelAnodeFrontAxisY.commands.enableAxis := FALSE;
       "Unit1.Em6.HmiInterface".cmMendrelAnodeFrontAxisY.commands.enableAxis := TRUE;
       "Unit1.Em6.ControlNodes".cmMendrelAnodeFrontAxisZ.commands.enableAxis := FALSE;
       "Unit1.Em6.HmiInterface".cmMendrelAnodeFrontAxisZ.commands.enableAxis := TRUE;
       "Unit1.Em6.ControlNodes".cmMendrelAnodeRearAxisY.commands.enableAxis := FALSE;
       "Unit1.Em6.HmiInterface".cmMendrelAnodeRearAxisY.commands.enableAxis := TRUE;
       "Unit1.Em6.ControlNodes".cmMendrelAnodeRearAxisZ.commands.enableAxis := FALSE;
       "Unit1.Em6.HmiInterface".cmMendrelAnodeRearAxisZ.commands.enableAxis := TRUE;
       "Unit1.Em6.ControlNodes".cmMendrelCathodeFrontAxisY.commands.enableAxis := FALSE;
       "Unit1.Em6.HmiInterface".cmMendrelCathodeFrontAxisY.commands.enableAxis := TRUE;
       "Unit1.Em6.ControlNodes".cmMendrelCathodeFrontAxisZ.commands.enableAxis := FALSE;
       "Unit1.Em6.HmiInterface".cmMendrelCathodeFrontAxisZ.commands.enableAxis := TRUE;
       "Unit1.Em6.ControlNodes".cmMendrelCathodeRearAxisY.commands.enableAxis := FALSE;
       "Unit1.Em6.HmiInterface".cmMendrelCathodeRearAxisY.commands.enableAxis := TRUE;
       "Unit1.Em6.ControlNodes".cmMendrelCathodeRearAxisZ.commands.enableAxis := FALSE;
       "Unit1.Em6.HmiInterface".cmMendrelCathodeRearAxisZ.commands.enableAxis := TRUE;
       "Unit1.Em6.ControlNodes".cmStackTableAxisZ.commands.enableAxis := FALSE;
       "Unit1.Em6.HmiInterface".cmStackTableAxisZ.commands.enableAxis := TRUE;
       "Unit1.Em6.ControlNodes".cmStackTableOutFrontAxisZ.commands.enableAxis := FALSE;
       "Unit1.Em6.HmiInterface".cmStackTableOutFrontAxisZ.commands.enableAxis := TRUE;
       "Unit1.Em6.ControlNodes".cmStackTableOutRearAxisZ.commands.enableAxis := FALSE;
       "Unit1.Em6.HmiInterface".cmStackTableOutRearAxisZ.commands.enableAxis := TRUE;
   END_IF;
   IF "Unit1.EmNodes".AllSFDoorOpen AND "Unit1.EmNodes".SS1TimeExtension THEN
       "Unit1.Em6.HmiInterface".cmFinalRollerFrontAxisX.commands.enableAxis := FALSE;
       "Unit1.Em6.ControlNodes".cmFinalRollerFrontAxisX.commands.enableAxis := TRUE;
       "Unit1.Em6.HmiInterface".cmFinalRollerRearAxisX.commands.enableAxis := FALSE;
       "Unit1.Em6.ControlNodes".cmFinalRollerRearAxisX.commands.enableAxis := TRUE;
       "Unit1.Em6.HmiInterface".cmMendrelAnodeFrontAxisY.commands.enableAxis := FALSE;
       "Unit1.Em6.ControlNodes".cmMendrelAnodeFrontAxisY.commands.enableAxis := TRUE;
       "Unit1.Em6.HmiInterface".cmMendrelAnodeFrontAxisZ.commands.enableAxis := FALSE;
       "Unit1.Em6.ControlNodes".cmMendrelAnodeFrontAxisZ.commands.enableAxis := TRUE;
       "Unit1.Em6.HmiInterface".cmMendrelAnodeRearAxisY.commands.enableAxis := FALSE;
       "Unit1.Em6.ControlNodes".cmMendrelAnodeRearAxisY.commands.enableAxis := TRUE;
       "Unit1.Em6.HmiInterface".cmMendrelAnodeRearAxisZ.commands.enableAxis := FALSE;
       "Unit1.Em6.ControlNodes".cmMendrelAnodeRearAxisZ.commands.enableAxis := TRUE;
       "Unit1.Em6.HmiInterface".cmMendrelCathodeFrontAxisY.commands.enableAxis := FALSE;
       "Unit1.Em6.ControlNodes".cmMendrelCathodeFrontAxisY.commands.enableAxis := TRUE;
       "Unit1.Em6.HmiInterface".cmMendrelCathodeFrontAxisZ.commands.enableAxis := FALSE;
       "Unit1.Em6.ControlNodes".cmMendrelCathodeFrontAxisZ.commands.enableAxis := TRUE;
       "Unit1.Em6.HmiInterface".cmMendrelCathodeRearAxisY.commands.enableAxis := FALSE;
       "Unit1.Em6.ControlNodes".cmMendrelCathodeRearAxisY.commands.enableAxis := TRUE;
       "Unit1.Em6.HmiInterface".cmMendrelCathodeRearAxisZ.commands.enableAxis := FALSE;
       "Unit1.Em6.ControlNodes".cmMendrelCathodeRearAxisZ.commands.enableAxis := TRUE;
       "Unit1.Em6.HmiInterface".cmStackTableAxisZ.commands.enableAxis := FALSE;
       "Unit1.Em6.ControlNodes".cmStackTableAxisZ.commands.enableAxis := TRUE;
       "Unit1.Em6.HmiInterface".cmStackTableOutFrontAxisZ.commands.enableAxis := FALSE;
       "Unit1.Em6.ControlNodes".cmStackTableOutFrontAxisZ.commands.enableAxis := TRUE;
       "Unit1.Em6.HmiInterface".cmStackTableOutRearAxisZ.commands.enableAxis := FALSE;
       "Unit1.Em6.ControlNodes".cmStackTableOutRearAxisZ.commands.enableAxis := TRUE;
   END_IF;
   #_w3 := "Unit1.EmNodes".AllSFDoorOpen AND NOT "Unit1.EmNodes".SS1TimeExtension AND NOT "Unit1.EmNodes".scsMode.auto AND (("Unit1.EmNodes".MobilePanelPermissions AND NOT "Unit1.EmNodes".pHmiMode.enable) OR (NOT "Unit1.EmNodes".MobilePanelPermissions AND NOT "Unit1.EmNodes".mainOpMode.enable)) AND #statSlmStatus.running;
   #_w4 := #_w3 AND NOT #statPulse.axisEnable[5];   // rising edge
   #statPulse.axisEnable[5] := #_w3;
   IF #_w4 THEN
       "Unit1.Em6.ControlNodes".cmFinalRollerFrontAxisX.commands.enableAxis := FALSE;
       "Unit1.Em6.HmiInterface".cmFinalRollerFrontAxisX.commands.enableAxis := FALSE;
       "Unit1.Em6.ControlNodes".cmFinalRollerRearAxisX.commands.enableAxis := FALSE;
       "Unit1.Em6.HmiInterface".cmFinalRollerRearAxisX.commands.enableAxis := FALSE;
       "Unit1.Em6.ControlNodes".cmMendrelAnodeFrontAxisY.commands.enableAxis := FALSE;
       "Unit1.Em6.HmiInterface".cmMendrelAnodeFrontAxisY.commands.enableAxis := FALSE;
       "Unit1.Em6.ControlNodes".cmMendrelAnodeFrontAxisZ.commands.enableAxis := FALSE;
       "Unit1.Em6.HmiInterface".cmMendrelAnodeFrontAxisZ.commands.enableAxis := FALSE;
       "Unit1.Em6.ControlNodes".cmMendrelAnodeRearAxisY.commands.enableAxis := FALSE;
       "Unit1.Em6.HmiInterface".cmMendrelAnodeRearAxisY.commands.enableAxis := FALSE;
       "Unit1.Em6.ControlNodes".cmMendrelAnodeRearAxisZ.commands.enableAxis := FALSE;
       "Unit1.Em6.HmiInterface".cmMendrelAnodeRearAxisZ.commands.enableAxis := FALSE;
       "Unit1.Em6.ControlNodes".cmMendrelCathodeFrontAxisY.commands.enableAxis := FALSE;
       "Unit1.Em6.HmiInterface".cmMendrelCathodeFrontAxisY.commands.enableAxis := FALSE;
       "Unit1.Em6.ControlNodes".cmMendrelCathodeFrontAxisZ.commands.enableAxis := FALSE;
       "Unit1.Em6.HmiInterface".cmMendrelCathodeFrontAxisZ.commands.enableAxis := FALSE;
       "Unit1.Em6.ControlNodes".cmMendrelCathodeRearAxisY.commands.enableAxis := FALSE;
       "Unit1.Em6.HmiInterface".cmMendrelCathodeRearAxisY.commands.enableAxis := FALSE;
       "Unit1.Em6.ControlNodes".cmMendrelCathodeRearAxisZ.commands.enableAxis := FALSE;
       "Unit1.Em6.HmiInterface".cmMendrelCathodeRearAxisZ.commands.enableAxis := FALSE;
       "Unit1.Em6.ControlNodes".cmStackTableAxisZ.commands.enableAxis := FALSE;
       "Unit1.Em6.HmiInterface".cmStackTableAxisZ.commands.enableAxis := FALSE;
       "Unit1.Em6.ControlNodes".cmStackTableOutFrontAxisZ.commands.enableAxis := FALSE;
       "Unit1.Em6.HmiInterface".cmStackTableOutFrontAxisZ.commands.enableAxis := FALSE;
       "Unit1.Em6.ControlNodes".cmStackTableOutRearAxisZ.commands.enableAxis := FALSE;
       "Unit1.Em6.HmiInterface".cmStackTableOutRearAxisZ.commands.enableAxis := FALSE;
   END_IF;
END_REGION

REGION Network 57: Disable All CMs
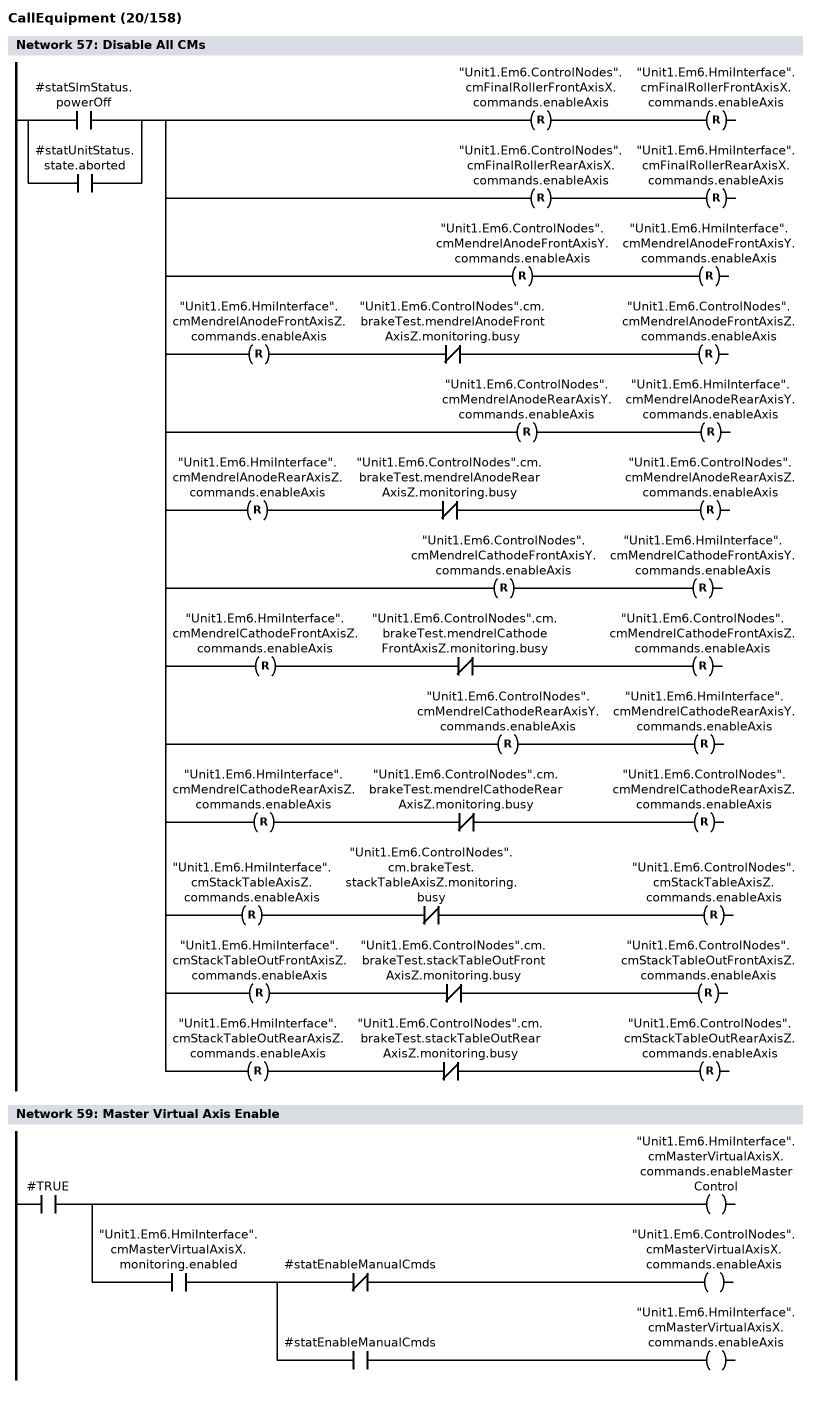
   RUNG wire#powerrail
      Contact( #statSlmStatus.powerOff )
      wire#w1
      R_Coil( "Unit1.Em6.ControlNodes".cmFinalRollerFrontAxisX.commands.enableAxis )
      R_Coil( "Unit1.Em6.HmiInterface".cmFinalRollerFrontAxisX.commands.enableAxis )
   END_RUNG
   RUNG wire#powerrail
      Contact( #statUnitStatus.state.aborted )
   END_RUNG wire#w1
   RUNG wire#w1
      R_Coil( "Unit1.Em6.ControlNodes".cmFinalRollerRearAxisX.commands.enableAxis )
      R_Coil( "Unit1.Em6.HmiInterface".cmFinalRollerRearAxisX.commands.enableAxis )
   END_RUNG
   RUNG wire#w1
      R_Coil( "Unit1.Em6.ControlNodes".cmMendrelAnodeFrontAxisY.commands.enableAxis )
      R_Coil( "Unit1.Em6.HmiInterface".cmMendrelAnodeFrontAxisY.commands.enableAxis )
   END_RUNG
   RUNG wire#w1
      R_Coil( "Unit1.Em6.HmiInterface".cmMendrelAnodeFrontAxisZ.commands.enableAxis )
      I_Contact( "Unit1.Em6.ControlNodes".cm.brakeTest.mendrelAnodeFrontAxisZ.monitoring.busy )
      R_Coil( "Unit1.Em6.ControlNodes".cmMendrelAnodeFrontAxisZ.commands.enableAxis )
   END_RUNG
   RUNG wire#w1
      R_Coil( "Unit1.Em6.ControlNodes".cmMendrelAnodeRearAxisY.commands.enableAxis )
      R_Coil( "Unit1.Em6.HmiInterface".cmMendrelAnodeRearAxisY.commands.enableAxis )
   END_RUNG
   RUNG wire#w1
      R_Coil( "Unit1.Em6.HmiInterface".cmMendrelAnodeRearAxisZ.commands.enableAxis )
      I_Contact( "Unit1.Em6.ControlNodes".cm.brakeTest.mendrelAnodeRearAxisZ.monitoring.busy )
      R_Coil( "Unit1.Em6.ControlNodes".cmMendrelAnodeRearAxisZ.commands.enableAxis )
   END_RUNG
   RUNG wire#w1
      R_Coil( "Unit1.Em6.ControlNodes".cmMendrelCathodeFrontAxisY.commands.enableAxis )
      R_Coil( "Unit1.Em6.HmiInterface".cmMendrelCathodeFrontAxisY.commands.enableAxis )
   END_RUNG
   RUNG wire#w1
      R_Coil( "Unit1.Em6.HmiInterface".cmMendrelCathodeFrontAxisZ.commands.enableAxis )
      I_Contact( "Unit1.Em6.ControlNodes".cm.brakeTest.mendrelCathodeFrontAxisZ.monitoring.busy )
      R_Coil( "Unit1.Em6.ControlNodes".cmMendrelCathodeFrontAxisZ.commands.enableAxis )
   END_RUNG
   RUNG wire#w1
      R_Coil( "Unit1.Em6.ControlNodes".cmMendrelCathodeRearAxisY.commands.enableAxis )
      R_Coil( "Unit1.Em6.HmiInterface".cmMendrelCathodeRearAxisY.commands.enableAxis )
   END_RUNG
   RUNG wire#w1
      R_Coil( "Unit1.Em6.HmiInterface".cmMendrelCathodeRearAxisZ.commands.enableAxis )
      I_Contact( "Unit1.Em6.ControlNodes".cm.brakeTest.mendrelCathodeRearAxisZ.monitoring.busy )
      R_Coil( "Unit1.Em6.ControlNodes".cmMendrelCathodeRearAxisZ.commands.enableAxis )
   END_RUNG
   RUNG wire#w1
      R_Coil( "Unit1.Em6.HmiInterface".cmStackTableAxisZ.commands.enableAxis )
      I_Contact( "Unit1.Em6.ControlNodes".cm.brakeTest.stackTableAxisZ.monitoring.busy )
      R_Coil( "Unit1.Em6.ControlNodes".cmStackTableAxisZ.commands.enableAxis )
   END_RUNG
   RUNG wire#w1
      R_Coil( "Unit1.Em6.HmiInterface".cmStackTableOutFrontAxisZ.commands.enableAxis )
      I_Contact( "Unit1.Em6.ControlNodes".cm.brakeTest.stackTableOutFrontAxisZ.monitoring.busy )
      R_Coil( "Unit1.Em6.ControlNodes".cmStackTableOutFrontAxisZ.commands.enableAxis )
   END_RUNG
   RUNG wire#w1
      R_Coil( "Unit1.Em6.HmiInterface".cmStackTableOutRearAxisZ.commands.enableAxis )
      I_Contact( "Unit1.Em6.ControlNodes".cm.brakeTest.stackTableOutRearAxisZ.monitoring.busy )
      R_Coil( "Unit1.Em6.ControlNodes".cmStackTableOutRearAxisZ.commands.enableAxis )
   END_RUNG
   // the same network as SCL:
   #_w1 := #statSlmStatus.powerOff OR #statUnitStatus.state.aborted;
   IF #_w1 THEN
       "Unit1.Em6.ControlNodes".cmFinalRollerFrontAxisX.commands.enableAxis := FALSE;
       "Unit1.Em6.HmiInterface".cmFinalRollerFrontAxisX.commands.enableAxis := FALSE;
       "Unit1.Em6.ControlNodes".cmFinalRollerRearAxisX.commands.enableAxis := FALSE;
       "Unit1.Em6.HmiInterface".cmFinalRollerRearAxisX.commands.enableAxis := FALSE;
       "Unit1.Em6.ControlNodes".cmMendrelAnodeFrontAxisY.commands.enableAxis := FALSE;
       "Unit1.Em6.HmiInterface".cmMendrelAnodeFrontAxisY.commands.enableAxis := FALSE;
       "Unit1.Em6.HmiInterface".cmMendrelAnodeFrontAxisZ.commands.enableAxis := FALSE;
   END_IF;
   IF #_w1 AND NOT "Unit1.Em6.ControlNodes".cm.brakeTest.mendrelAnodeFrontAxisZ.monitoring.busy THEN
       "Unit1.Em6.ControlNodes".cmMendrelAnodeFrontAxisZ.commands.enableAxis := FALSE;
   END_IF;
   IF #_w1 THEN
       "Unit1.Em6.ControlNodes".cmMendrelAnodeRearAxisY.commands.enableAxis := FALSE;
       "Unit1.Em6.HmiInterface".cmMendrelAnodeRearAxisY.commands.enableAxis := FALSE;
       "Unit1.Em6.HmiInterface".cmMendrelAnodeRearAxisZ.commands.enableAxis := FALSE;
   END_IF;
   IF #_w1 AND NOT "Unit1.Em6.ControlNodes".cm.brakeTest.mendrelAnodeRearAxisZ.monitoring.busy THEN
       "Unit1.Em6.ControlNodes".cmMendrelAnodeRearAxisZ.commands.enableAxis := FALSE;
   END_IF;
   IF #_w1 THEN
       "Unit1.Em6.ControlNodes".cmMendrelCathodeFrontAxisY.commands.enableAxis := FALSE;
       "Unit1.Em6.HmiInterface".cmMendrelCathodeFrontAxisY.commands.enableAxis := FALSE;
       "Unit1.Em6.HmiInterface".cmMendrelCathodeFrontAxisZ.commands.enableAxis := FALSE;
   END_IF;
   IF #_w1 AND NOT "Unit1.Em6.ControlNodes".cm.brakeTest.mendrelCathodeFrontAxisZ.monitoring.busy THEN
       "Unit1.Em6.ControlNodes".cmMendrelCathodeFrontAxisZ.commands.enableAxis := FALSE;
   END_IF;
   IF #_w1 THEN
       "Unit1.Em6.ControlNodes".cmMendrelCathodeRearAxisY.commands.enableAxis := FALSE;
       "Unit1.Em6.HmiInterface".cmMendrelCathodeRearAxisY.commands.enableAxis := FALSE;
       "Unit1.Em6.HmiInterface".cmMendrelCathodeRearAxisZ.commands.enableAxis := FALSE;
   END_IF;
   IF #_w1 AND NOT "Unit1.Em6.ControlNodes".cm.brakeTest.mendrelCathodeRearAxisZ.monitoring.busy THEN
       "Unit1.Em6.ControlNodes".cmMendrelCathodeRearAxisZ.commands.enableAxis := FALSE;
   END_IF;
   IF #_w1 THEN "Unit1.Em6.HmiInterface".cmStackTableAxisZ.commands.enableAxis := FALSE; END_IF;
   IF #_w1 AND NOT "Unit1.Em6.ControlNodes".cm.brakeTest.stackTableAxisZ.monitoring.busy THEN
       "Unit1.Em6.ControlNodes".cmStackTableAxisZ.commands.enableAxis := FALSE;
   END_IF;
   IF #_w1 THEN "Unit1.Em6.HmiInterface".cmStackTableOutFrontAxisZ.commands.enableAxis := FALSE; END_IF;
   IF #_w1 AND NOT "Unit1.Em6.ControlNodes".cm.brakeTest.stackTableOutFrontAxisZ.monitoring.busy THEN
       "Unit1.Em6.ControlNodes".cmStackTableOutFrontAxisZ.commands.enableAxis := FALSE;
   END_IF;
   IF #_w1 THEN "Unit1.Em6.HmiInterface".cmStackTableOutRearAxisZ.commands.enableAxis := FALSE; END_IF;
   IF #_w1 AND NOT "Unit1.Em6.ControlNodes".cm.brakeTest.stackTableOutRearAxisZ.monitoring.busy THEN
       "Unit1.Em6.ControlNodes".cmStackTableOutRearAxisZ.commands.enableAxis := FALSE;
   END_IF;
END_REGION

REGION Network 59: Master Virtual Axis Enable
   RUNG wire#powerrail
      Contact( #TRUE )
      wire#w1
      Coil( "Unit1.Em6.HmiInterface".cmMasterVirtualAxisX.commands.enableMasterControl )
   END_RUNG
   RUNG wire#w1
      Contact( "Unit1.Em6.HmiInterface".cmMasterVirtualAxisX.monitoring.enabled )
      wire#w2
      I_Contact( #statEnableManualCmds )
      Coil( "Unit1.Em6.ControlNodes".cmMasterVirtualAxisX.commands.enableAxis )
   END_RUNG
   RUNG wire#w2
      Contact( #statEnableManualCmds )
      Coil( "Unit1.Em6.HmiInterface".cmMasterVirtualAxisX.commands.enableAxis )
   END_RUNG
   // the same network as SCL:
   "Unit1.Em6.HmiInterface".cmMasterVirtualAxisX.commands.enableMasterControl := #TRUE;
   #_w1 := #TRUE AND "Unit1.Em6.HmiInterface".cmMasterVirtualAxisX.monitoring.enabled;
   "Unit1.Em6.ControlNodes".cmMasterVirtualAxisX.commands.enableAxis := #_w1 AND NOT #statEnableManualCmds;
   "Unit1.Em6.HmiInterface".cmMasterVirtualAxisX.commands.enableAxis := #_w1 AND #statEnableManualCmds;
END_REGION

REGION Network 60: Master Virtual Axis Homing
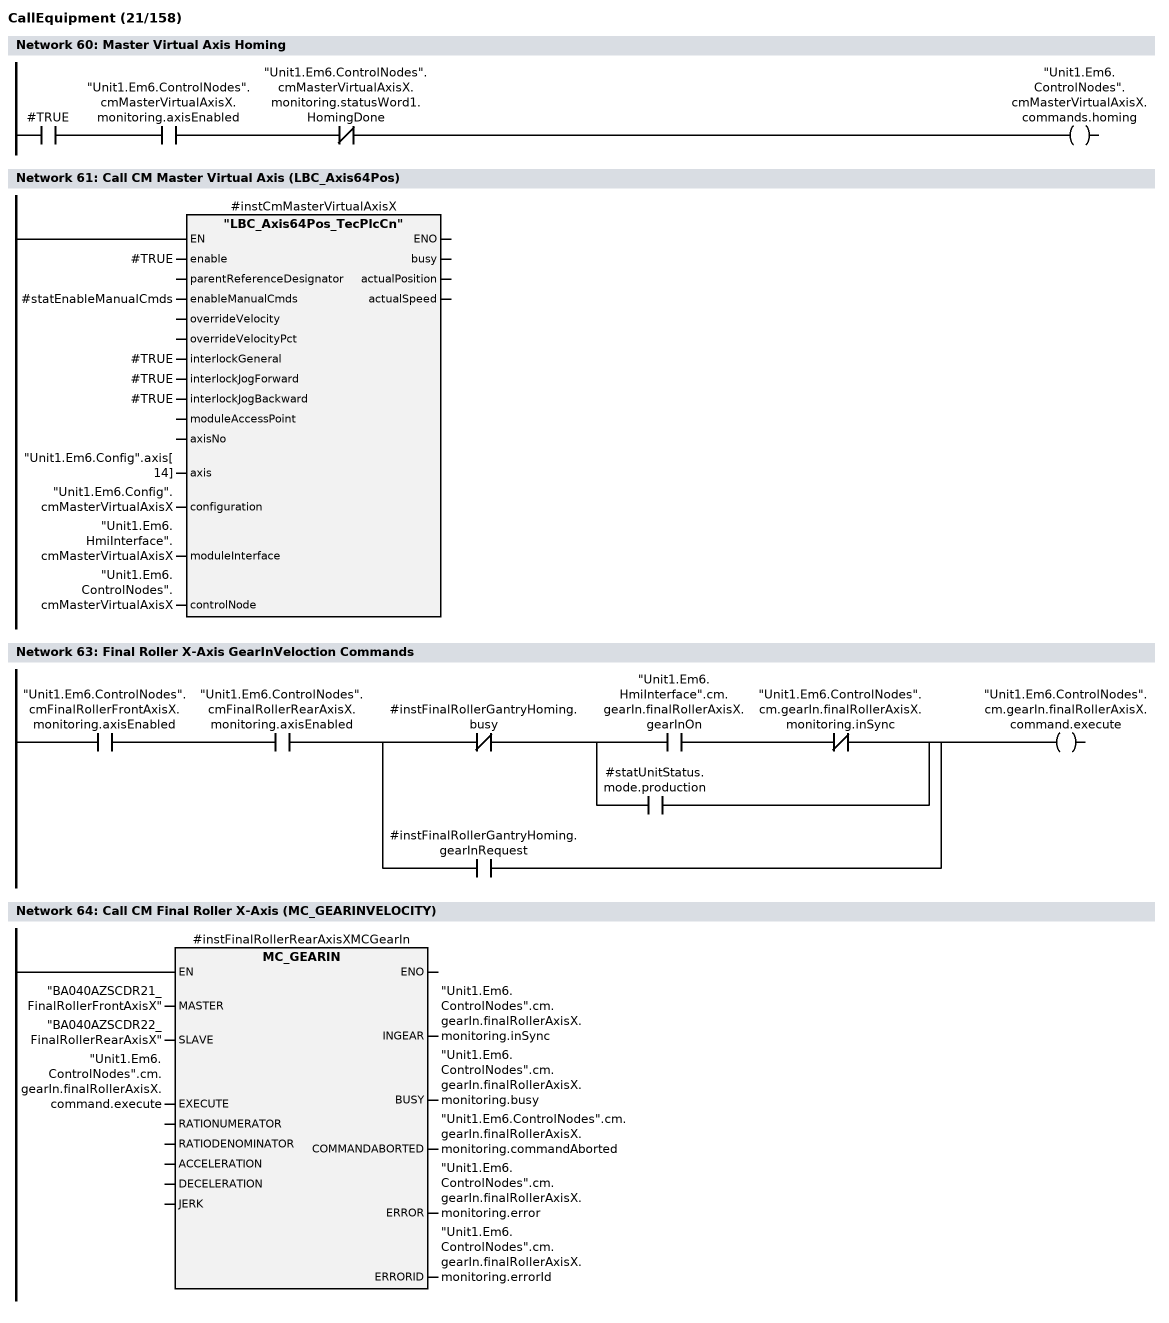
   RUNG wire#powerrail
      Contact( #TRUE )
      Contact( "Unit1.Em6.ControlNodes".cmMasterVirtualAxisX.monitoring.axisEnabled )
      I_Contact( "Unit1.Em6.ControlNodes".cmMasterVirtualAxisX.monitoring.statusWord1.HomingDone )
      Coil( "Unit1.Em6.ControlNodes".cmMasterVirtualAxisX.commands.homing )
   END_RUNG
   // the same network as SCL:
   "Unit1.Em6.ControlNodes".cmMasterVirtualAxisX.commands.homing := #TRUE AND "Unit1.Em6.ControlNodes".cmMasterVirtualAxisX.monitoring.axisEnabled AND NOT "Unit1.Em6.ControlNodes".cmMasterVirtualAxisX.monitoring.statusWord1.HomingDone;
END_REGION

REGION Network 61: Call CM Master Virtual Axis (LBC_Axis64Pos)
   RUNG wire#powerrail
      #instCmMasterVirtualAxisX(enable := #TRUE, parentReferenceDesignator :=, enableManualCmds := #statEnableManualCmds, overrideVelocity :=, overrideVelocityPct :=, interlockGeneral := #TRUE, interlockJogForward := #TRUE, interlockJogBackward := #TRUE, moduleAccessPoint :=, axisNo :=, axis := "Unit1.Em6.Config".axis[14], configuration := "Unit1.Em6.Config".cmMasterVirtualAxisX, moduleInterface := "Unit1.Em6.HmiInterface".cmMasterVirtualAxisX, controlNode := "Unit1.Em6.ControlNodes".cmMasterVirtualAxisX, busy =>, actualPosition =>, actualSpeed =>)
   END_RUNG
   // the same network as SCL:
   #instCmMasterVirtualAxisX(enable := #TRUE,   // "LBC_Axis64Pos_TecPlcCn"
                           enableManualCmds := #statEnableManualCmds,
                           interlockGeneral := #TRUE,
                           interlockJogForward := #TRUE,
                           interlockJogBackward := #TRUE,
                           axis := "Unit1.Em6.Config".axis[14],
                           configuration := "Unit1.Em6.Config".cmMasterVirtualAxisX,
                           moduleInterface := "Unit1.Em6.HmiInterface".cmMasterVirtualAxisX,
                           controlNode := "Unit1.Em6.ControlNodes".cmMasterVirtualAxisX);
END_REGION

REGION Network 63: Final Roller X-Axis GearInVeloction Commands
   RUNG wire#powerrail
      Contact( "Unit1.Em6.ControlNodes".cmFinalRollerFrontAxisX.monitoring.axisEnabled )
      Contact( "Unit1.Em6.ControlNodes".cmFinalRollerRearAxisX.monitoring.axisEnabled )
      wire#w1
      I_Contact( #instFinalRollerGantryHoming.busy )
      wire#w2
      Contact( "Unit1.Em6.HmiInterface".cm.gearIn.finalRollerAxisX.gearInOn )
      I_Contact( "Unit1.Em6.ControlNodes".cm.gearIn.finalRollerAxisX.monitoring.inSync )
      wire#w3
      Coil( "Unit1.Em6.ControlNodes".cm.gearIn.finalRollerAxisX.command.execute )
   END_RUNG
   RUNG wire#w2
      Contact( #statUnitStatus.mode.production )
   END_RUNG wire#w3
   RUNG wire#w1
      Contact( #instFinalRollerGantryHoming.gearInRequest )
   END_RUNG wire#w3
   // the same network as SCL:
   "Unit1.Em6.ControlNodes".cm.gearIn.finalRollerAxisX.command.execute := "Unit1.Em6.ControlNodes".cmFinalRollerFrontAxisX.monitoring.axisEnabled AND "Unit1.Em6.ControlNodes".cmFinalRollerRearAxisX.monitoring.axisEnabled AND ((NOT #instFinalRollerGantryHoming.busy AND (("Unit1.Em6.HmiInterface".cm.gearIn.finalRollerAxisX.gearInOn AND NOT "Unit1.Em6.ControlNodes".cm.gearIn.finalRollerAxisX.monitoring.inSync) OR #statUnitStatus.mode.production)) OR #instFinalRollerGantryHoming.gearInRequest);
END_REGION

REGION Network 64: Call CM Final Roller X-Axis (MC_GEARINVELOCITY)
   RUNG wire#powerrail
      #instFinalRollerRearAxisXMCGearIn.MC_GEARIN(Master := "BA040AZSCDR21_FinalRollerFrontAxisX", Slave := "BA040AZSCDR22_FinalRollerRearAxisX", Execute := "Unit1.Em6.ControlNodes".cm.gearIn.finalRollerAxisX.command.execute, RatioNumerator :=, RatioDenominator :=, Acceleration :=, Deceleration :=, Jerk :=, InGear => "Unit1.Em6.ControlNodes".cm.gearIn.finalRollerAxisX.monitoring.inSync, Busy => "Unit1.Em6.ControlNodes".cm.gearIn.finalRollerAxisX.monitoring.busy, CommandAborted => "Unit1.Em6.ControlNodes".cm.gearIn.finalRollerAxisX.monitoring.commandAborted, Error => "Unit1.Em6.ControlNodes".cm.gearIn.finalRollerAxisX.monitoring.error, ErrorId => "Unit1.Em6.ControlNodes".cm.gearIn.finalRollerAxisX.monitoring.errorId)
   END_RUNG
   // the same network as SCL:
   #instFinalRollerRearAxisXMCGearIn(Master := "BA040AZSCDR21_FinalRollerFrontAxisX",   // MC_GEARIN
                           Slave := "BA040AZSCDR22_FinalRollerRearAxisX",
                           Execute := "Unit1.Em6.ControlNodes".cm.gearIn.finalRollerAxisX.command.execute,
                           InGear => "Unit1.Em6.ControlNodes".cm.gearIn.finalRollerAxisX.monitoring.inSync,
                           Busy => "Unit1.Em6.ControlNodes".cm.gearIn.finalRollerAxisX.monitoring.busy,
                           CommandAborted => "Unit1.Em6.ControlNodes".cm.gearIn.finalRollerAxisX.monitoring.commandAborted,
                           Error => "Unit1.Em6.ControlNodes".cm.gearIn.finalRollerAxisX.monitoring.error,
                           ErrorId => "Unit1.Em6.ControlNodes".cm.gearIn.finalRollerAxisX.monitoring.errorId);
END_REGION

REGION Network 65: Call CM Final Roller X-Axis (LER_GantryHoming)
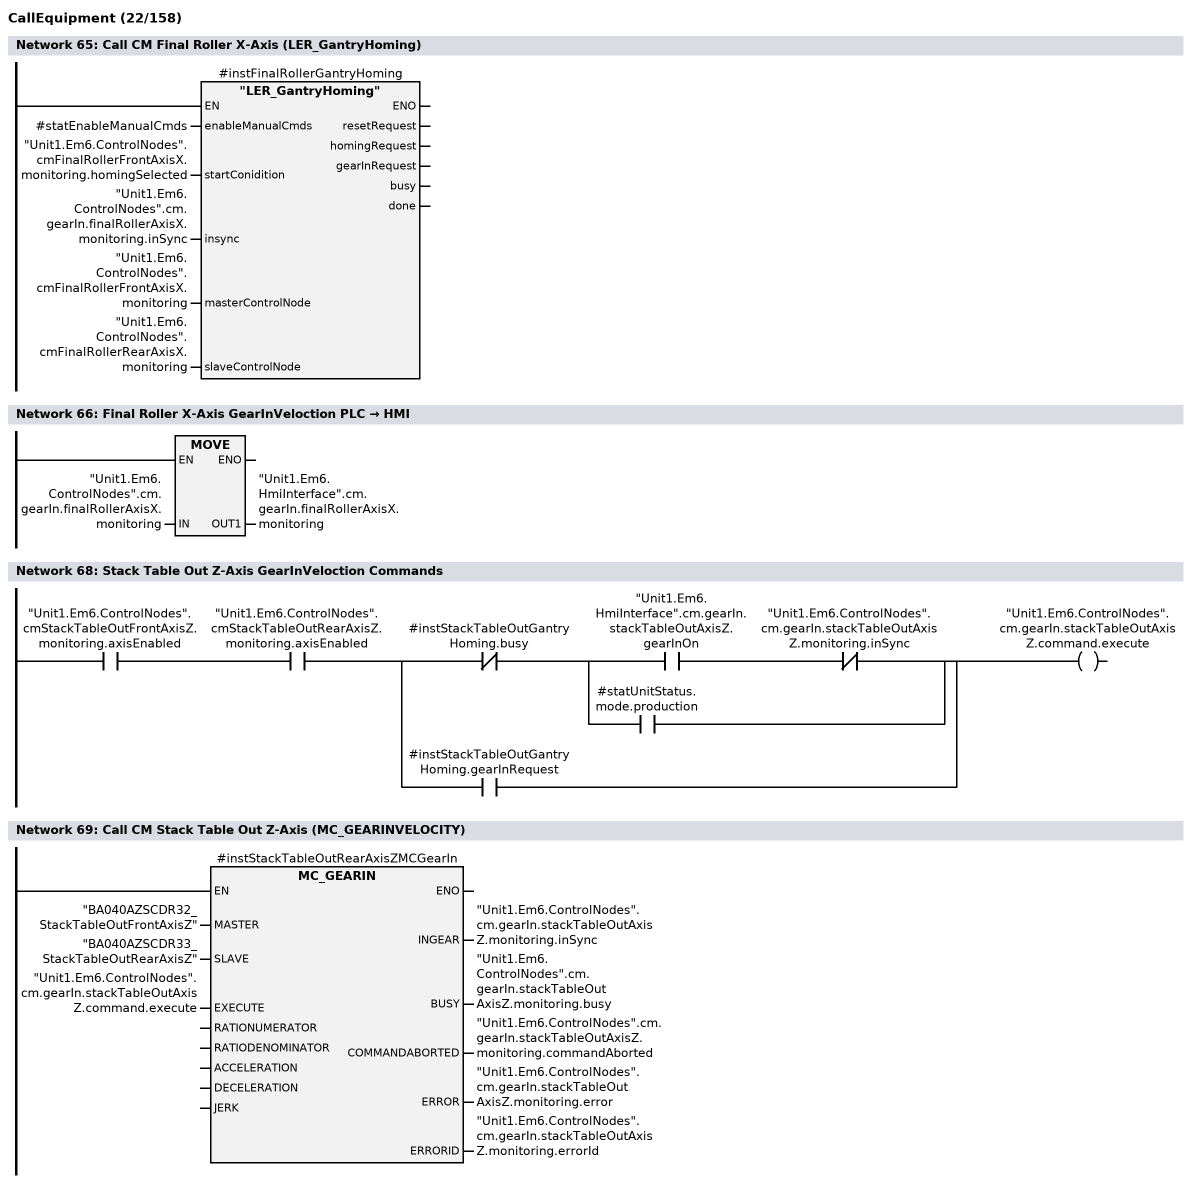
   RUNG wire#powerrail
      #instFinalRollerGantryHoming(enableManualCmds := #statEnableManualCmds, startConidition := "Unit1.Em6.ControlNodes".cmFinalRollerFrontAxisX.monitoring.homingSelected, insync := "Unit1.Em6.ControlNodes".cm.gearIn.finalRollerAxisX.monitoring.inSync, masterControlNode := "Unit1.Em6.ControlNodes".cmFinalRollerFrontAxisX.monitoring, slaveControlNode := "Unit1.Em6.ControlNodes".cmFinalRollerRearAxisX.monitoring, resetRequest =>, homingRequest =>, gearInRequest =>, busy =>, done =>)
   END_RUNG
   // the same network as SCL:
   #instFinalRollerGantryHoming(enableManualCmds := #statEnableManualCmds,   // "LER_GantryHoming"
                           startConidition := "Unit1.Em6.ControlNodes".cmFinalRollerFrontAxisX.monitoring.homingSelected,
                           insync := "Unit1.Em6.ControlNodes".cm.gearIn.finalRollerAxisX.monitoring.inSync,
                           masterControlNode := "Unit1.Em6.ControlNodes".cmFinalRollerFrontAxisX.monitoring,
                           slaveControlNode := "Unit1.Em6.ControlNodes".cmFinalRollerRearAxisX.monitoring);
END_REGION

REGION Network 66: Final Roller X-Axis GearInVeloction PLC → HMI
   RUNG wire#powerrail
      Move(in := "Unit1.Em6.ControlNodes".cm.gearIn.finalRollerAxisX.monitoring, out1 => "Unit1.Em6.HmiInterface".cm.gearIn.finalRollerAxisX.monitoring)
   END_RUNG
   // the same network as SCL:
   "Unit1.Em6.HmiInterface".cm.gearIn.finalRollerAxisX.monitoring := "Unit1.Em6.ControlNodes".cm.gearIn.finalRollerAxisX.monitoring;
END_REGION

REGION Network 68: Stack Table Out Z-Axis GearInVeloction Commands
   RUNG wire#powerrail
      Contact( "Unit1.Em6.ControlNodes".cmStackTableOutFrontAxisZ.monitoring.axisEnabled )
      Contact( "Unit1.Em6.ControlNodes".cmStackTableOutRearAxisZ.monitoring.axisEnabled )
      wire#w1
      I_Contact( #instStackTableOutGantryHoming.busy )
      wire#w2
      Contact( "Unit1.Em6.HmiInterface".cm.gearIn.stackTableOutAxisZ.gearInOn )
      I_Contact( "Unit1.Em6.ControlNodes".cm.gearIn.stackTableOutAxisZ.monitoring.inSync )
      wire#w3
      Coil( "Unit1.Em6.ControlNodes".cm.gearIn.stackTableOutAxisZ.command.execute )
   END_RUNG
   RUNG wire#w2
      Contact( #statUnitStatus.mode.production )
   END_RUNG wire#w3
   RUNG wire#w1
      Contact( #instStackTableOutGantryHoming.gearInRequest )
   END_RUNG wire#w3
   // the same network as SCL:
   "Unit1.Em6.ControlNodes".cm.gearIn.stackTableOutAxisZ.command.execute := "Unit1.Em6.ControlNodes".cmStackTableOutFrontAxisZ.monitoring.axisEnabled AND "Unit1.Em6.ControlNodes".cmStackTableOutRearAxisZ.monitoring.axisEnabled AND ((NOT #instStackTableOutGantryHoming.busy AND (("Unit1.Em6.HmiInterface".cm.gearIn.stackTableOutAxisZ.gearInOn AND NOT "Unit1.Em6.ControlNodes".cm.gearIn.stackTableOutAxisZ.monitoring.inSync) OR #statUnitStatus.mode.production)) OR #instStackTableOutGantryHoming.gearInRequest);
END_REGION

REGION Network 69: Call CM Stack Table Out Z-Axis (MC_GEARINVELOCITY)
   RUNG wire#powerrail
      #instStackTableOutRearAxisZMCGearIn.MC_GEARIN(Master := "BA040AZSCDR32_StackTableOutFrontAxisZ", Slave := "BA040AZSCDR33_StackTableOutRearAxisZ", Execute := "Unit1.Em6.ControlNodes".cm.gearIn.stackTableOutAxisZ.command.execute, RatioNumerator :=, RatioDenominator :=, Acceleration :=, Deceleration :=, Jerk :=, InGear => "Unit1.Em6.ControlNodes".cm.gearIn.stackTableOutAxisZ.monitoring.inSync, Busy => "Unit1.Em6.ControlNodes".cm.gearIn.stackTableOutAxisZ.monitoring.busy, CommandAborted => "Unit1.Em6.ControlNodes".cm.gearIn.stackTableOutAxisZ.monitoring.commandAborted, Error => "Unit1.Em6.ControlNodes".cm.gearIn.stackTableOutAxisZ.monitoring.error, ErrorId => "Unit1.Em6.ControlNodes".cm.gearIn.stackTableOutAxisZ.monitoring.errorId)
   END_RUNG
   // the same network as SCL:
   #instStackTableOutRearAxisZMCGearIn(Master := "BA040AZSCDR32_StackTableOutFrontAxisZ",   // MC_GEARIN
                           Slave := "BA040AZSCDR33_StackTableOutRearAxisZ",
                           Execute := "Unit1.Em6.ControlNodes".cm.gearIn.stackTableOutAxisZ.command.execute,
                           InGear => "Unit1.Em6.ControlNodes".cm.gearIn.stackTableOutAxisZ.monitoring.inSync,
                           Busy => "Unit1.Em6.ControlNodes".cm.gearIn.stackTableOutAxisZ.monitoring.busy,
                           CommandAborted => "Unit1.Em6.ControlNodes".cm.gearIn.stackTableOutAxisZ.monitoring.commandAborted,
                           Error => "Unit1.Em6.ControlNodes".cm.gearIn.stackTableOutAxisZ.monitoring.error,
                           ErrorId => "Unit1.Em6.ControlNodes".cm.gearIn.stackTableOutAxisZ.monitoring.errorId);
END_REGION

REGION Network 70: Call CM Stack Table Out Z-Axis (LER_GantryHoming)
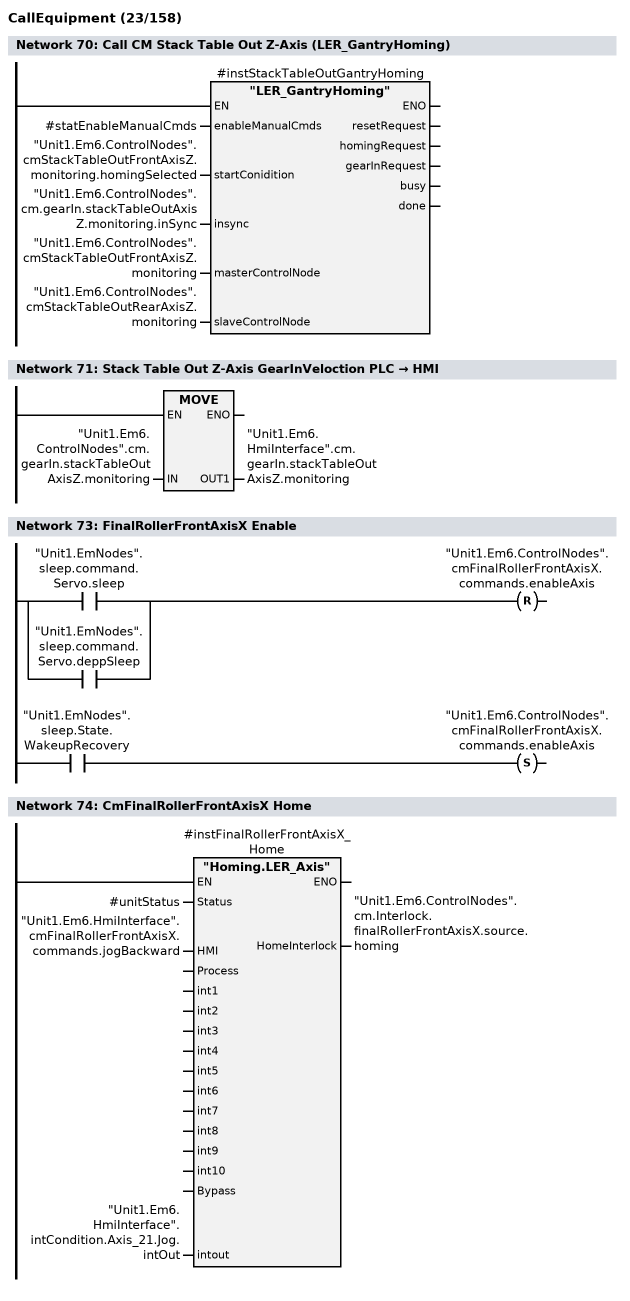
   RUNG wire#powerrail
      #instStackTableOutGantryHoming(enableManualCmds := #statEnableManualCmds, startConidition := "Unit1.Em6.ControlNodes".cmStackTableOutFrontAxisZ.monitoring.homingSelected, insync := "Unit1.Em6.ControlNodes".cm.gearIn.stackTableOutAxisZ.monitoring.inSync, masterControlNode := "Unit1.Em6.ControlNodes".cmStackTableOutFrontAxisZ.monitoring, slaveControlNode := "Unit1.Em6.ControlNodes".cmStackTableOutRearAxisZ.monitoring, resetRequest =>, homingRequest =>, gearInRequest =>, busy =>, done =>)
   END_RUNG
   // the same network as SCL:
   #instStackTableOutGantryHoming(enableManualCmds := #statEnableManualCmds,   // "LER_GantryHoming"
                           startConidition := "Unit1.Em6.ControlNodes".cmStackTableOutFrontAxisZ.monitoring.homingSelected,
                           insync := "Unit1.Em6.ControlNodes".cm.gearIn.stackTableOutAxisZ.monitoring.inSync,
                           masterControlNode := "Unit1.Em6.ControlNodes".cmStackTableOutFrontAxisZ.monitoring,
                           slaveControlNode := "Unit1.Em6.ControlNodes".cmStackTableOutRearAxisZ.monitoring);
END_REGION

REGION Network 71: Stack Table Out Z-Axis GearInVeloction PLC → HMI
   RUNG wire#powerrail
      Move(in := "Unit1.Em6.ControlNodes".cm.gearIn.stackTableOutAxisZ.monitoring, out1 => "Unit1.Em6.HmiInterface".cm.gearIn.stackTableOutAxisZ.monitoring)
   END_RUNG
   // the same network as SCL:
   "Unit1.Em6.HmiInterface".cm.gearIn.stackTableOutAxisZ.monitoring := "Unit1.Em6.ControlNodes".cm.gearIn.stackTableOutAxisZ.monitoring;
END_REGION

REGION Network 73: FinalRollerFrontAxisX Enable
   RUNG wire#powerrail
      Contact( "Unit1.EmNodes".sleep.command.Servo.sleep )
      wire#w1
      R_Coil( "Unit1.Em6.ControlNodes".cmFinalRollerFrontAxisX.commands.enableAxis )
   END_RUNG
   RUNG wire#powerrail
      Contact( "Unit1.EmNodes".sleep.command.Servo.deppSleep )
   END_RUNG wire#w1
   RUNG wire#powerrail
      Contact( "Unit1.EmNodes".sleep.State.WakeupRecovery )
      S_Coil( "Unit1.Em6.ControlNodes".cmFinalRollerFrontAxisX.commands.enableAxis )
   END_RUNG
   // the same network as SCL:
   IF "Unit1.EmNodes".sleep.command.Servo.sleep OR "Unit1.EmNodes".sleep.command.Servo.deppSleep THEN
       "Unit1.Em6.ControlNodes".cmFinalRollerFrontAxisX.commands.enableAxis := FALSE;
   END_IF;
   IF "Unit1.EmNodes".sleep.State.WakeupRecovery THEN
       "Unit1.Em6.ControlNodes".cmFinalRollerFrontAxisX.commands.enableAxis := TRUE;
   END_IF;
END_REGION

REGION Network 74: CmFinalRollerFrontAxisX Home
   RUNG wire#powerrail
      #instFinalRollerFrontAxisX_Home(Status := #unitStatus, HMI := "Unit1.Em6.HmiInterface".cmFinalRollerFrontAxisX.commands.jogBackward, Process :=, int1 :=, int2 :=, int3 :=, int4 :=, int5 :=, int6 :=, int7 :=, int8 :=, int9 :=, int10 :=, Bypass :=, intout := "Unit1.Em6.HmiInterface".intCondition.Axis_21.Jog.intOut, HomeInterlock => "Unit1.Em6.ControlNodes".cm.Interlock.finalRollerFrontAxisX.source.homing)
   END_RUNG
   // the same network as SCL:
   #instFinalRollerFrontAxisX_Home(Status := #unitStatus,   // "Homing.LER_Axis"
                           HMI := "Unit1.Em6.HmiInterface".cmFinalRollerFrontAxisX.commands.jogBackward,
                           intout := "Unit1.Em6.HmiInterface".intCondition.Axis_21.Jog.intOut,
                           HomeInterlock => "Unit1.Em6.ControlNodes".cm.Interlock.finalRollerFrontAxisX.source.homing);
END_REGION

REGION Network 75: CmFinalRollerFrontAxisX Position Absolute Jog
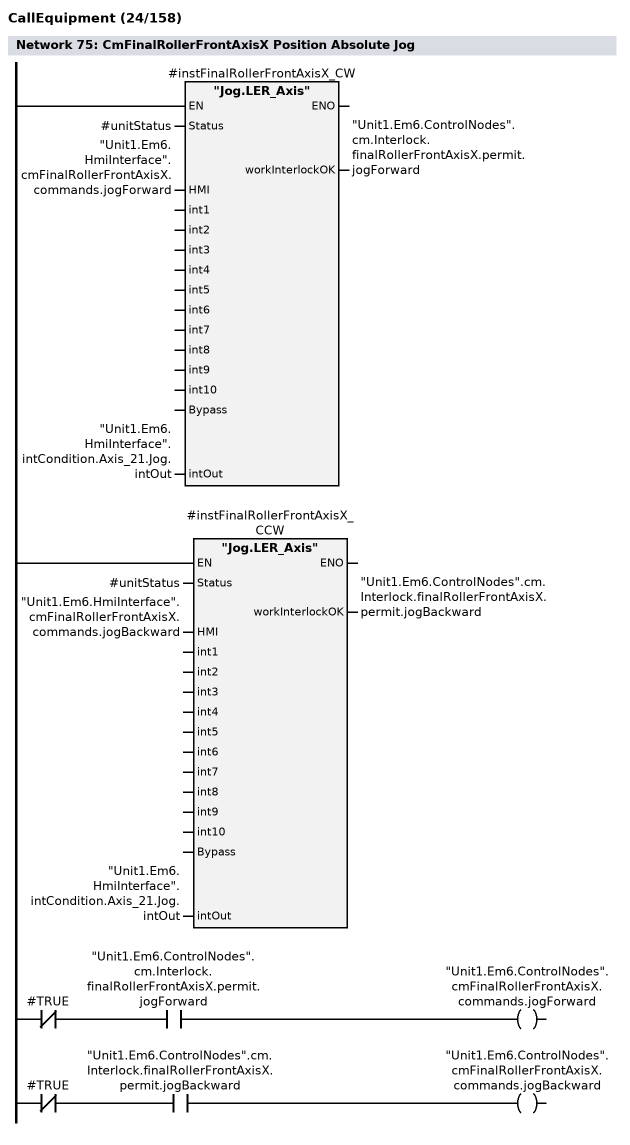
   RUNG wire#powerrail
      #instFinalRollerFrontAxisX_CW(Status := #unitStatus, HMI := "Unit1.Em6.HmiInterface".cmFinalRollerFrontAxisX.commands.jogForward, int1 :=, int2 :=, int3 :=, int4 :=, int5 :=, int6 :=, int7 :=, int8 :=, int9 :=, int10 :=, Bypass :=, intOut := "Unit1.Em6.HmiInterface".intCondition.Axis_21.Jog.intOut, workInterlockOK => "Unit1.Em6.ControlNodes".cm.Interlock.finalRollerFrontAxisX.permit.jogForward)
   END_RUNG
   RUNG wire#powerrail
      #instFinalRollerFrontAxisX_CCW(Status := #unitStatus, HMI := "Unit1.Em6.HmiInterface".cmFinalRollerFrontAxisX.commands.jogBackward, int1 :=, int2 :=, int3 :=, int4 :=, int5 :=, int6 :=, int7 :=, int8 :=, int9 :=, int10 :=, Bypass :=, intOut := "Unit1.Em6.HmiInterface".intCondition.Axis_21.Jog.intOut, workInterlockOK => "Unit1.Em6.ControlNodes".cm.Interlock.finalRollerFrontAxisX.permit.jogBackward)
   END_RUNG
   RUNG wire#powerrail
      I_Contact( #TRUE )
      Contact( "Unit1.Em6.ControlNodes".cm.Interlock.finalRollerFrontAxisX.permit.jogForward )
      Coil( "Unit1.Em6.ControlNodes".cmFinalRollerFrontAxisX.commands.jogForward )
   END_RUNG
   RUNG wire#powerrail
      I_Contact( #TRUE )
      Contact( "Unit1.Em6.ControlNodes".cm.Interlock.finalRollerFrontAxisX.permit.jogBackward )
      Coil( "Unit1.Em6.ControlNodes".cmFinalRollerFrontAxisX.commands.jogBackward )
   END_RUNG
   // the same network as SCL:
   #instFinalRollerFrontAxisX_CW(Status := #unitStatus,   // "Jog.LER_Axis"
                           HMI := "Unit1.Em6.HmiInterface".cmFinalRollerFrontAxisX.commands.jogForward,
                           intOut := "Unit1.Em6.HmiInterface".intCondition.Axis_21.Jog.intOut,
                           workInterlockOK => "Unit1.Em6.ControlNodes".cm.Interlock.finalRollerFrontAxisX.permit.jogForward);
   #instFinalRollerFrontAxisX_CCW(Status := #unitStatus,   // "Jog.LER_Axis"
                           HMI := "Unit1.Em6.HmiInterface".cmFinalRollerFrontAxisX.commands.jogBackward,
                           intOut := "Unit1.Em6.HmiInterface".intCondition.Axis_21.Jog.intOut,
                           workInterlockOK => "Unit1.Em6.ControlNodes".cm.Interlock.finalRollerFrontAxisX.permit.jogBackward);
   "Unit1.Em6.ControlNodes".cmFinalRollerFrontAxisX.commands.jogForward := NOT #TRUE AND "Unit1.Em6.ControlNodes".cm.Interlock.finalRollerFrontAxisX.permit.jogForward;
   "Unit1.Em6.ControlNodes".cmFinalRollerFrontAxisX.commands.jogBackward := NOT #TRUE AND "Unit1.Em6.ControlNodes".cm.Interlock.finalRollerFrontAxisX.permit.jogBackward;
END_REGION

REGION Network 76: CmFinalRollerFrontAxisX Position Absolute Position0
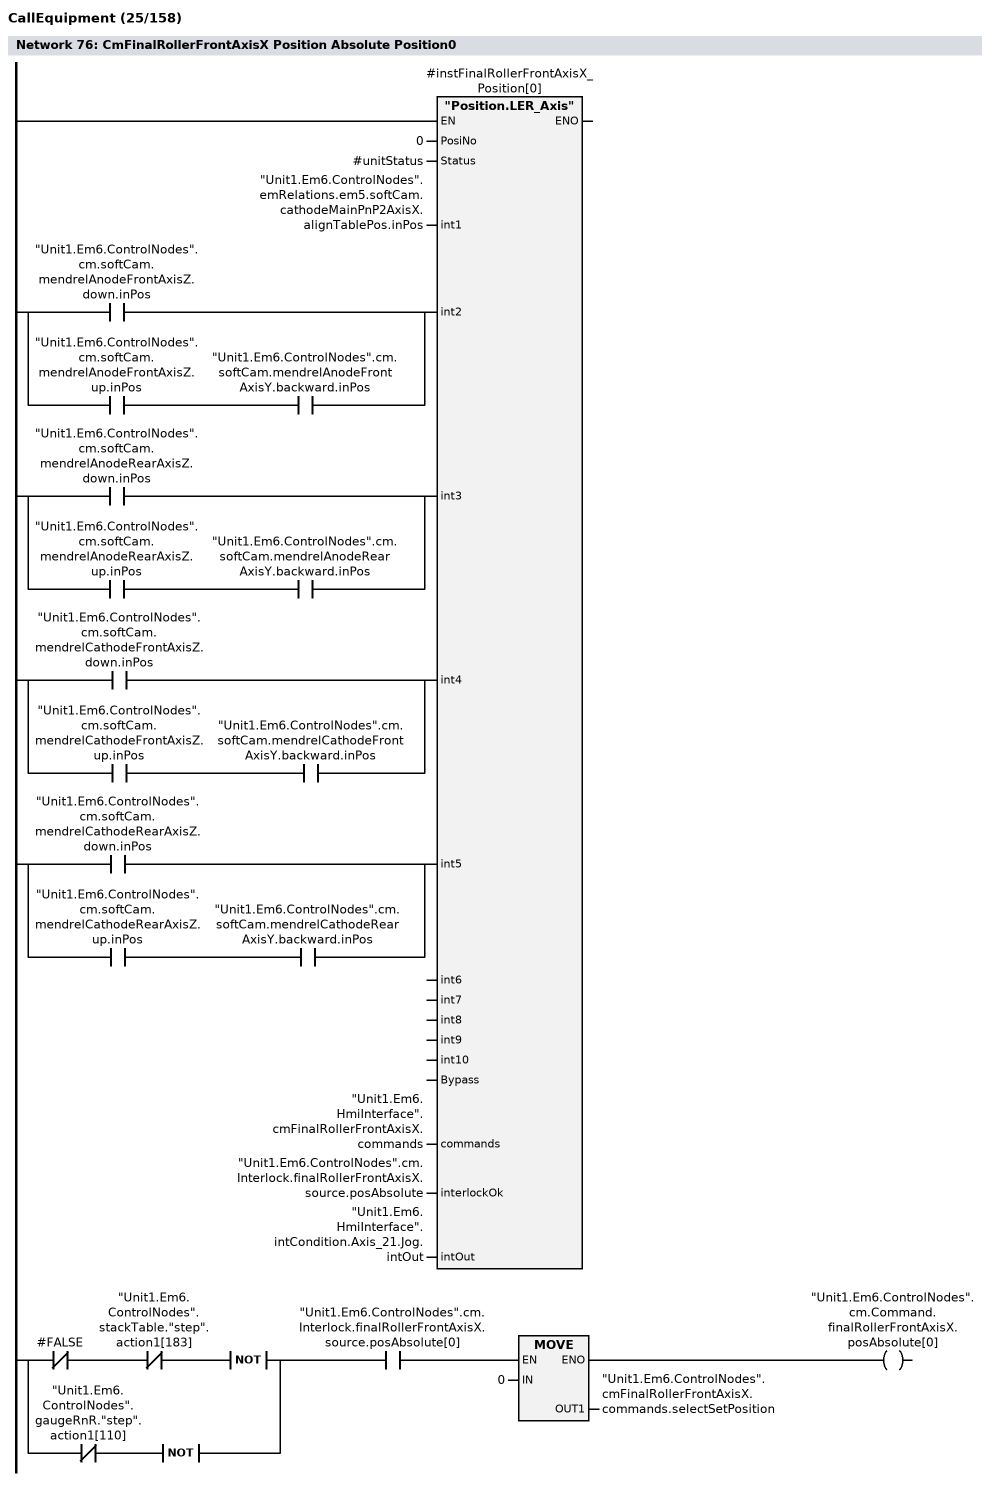
   RUNG wire#powerrail
      #instFinalRollerFrontAxisX_Position[0](int2 := wire#w1, int3 := wire#w2, int4 := wire#w3, int5 := wire#w4, PosiNo := 0, Status := #unitStatus, int1 := "Unit1.Em6.ControlNodes".emRelations.em5.softCam.cathodeMainPnP2AxisX.alignTablePos.inPos, int6 :=, int7 :=, int8 :=, int9 :=, int10 :=, Bypass :=, commands := "Unit1.Em6.HmiInterface".cmFinalRollerFrontAxisX.commands, interlockOk := "Unit1.Em6.ControlNodes".cm.Interlock.finalRollerFrontAxisX.source.posAbsolute, intOut := "Unit1.Em6.HmiInterface".intCondition.Axis_21.Jog.intOut)
   END_RUNG
   RUNG wire#powerrail
      Contact( "Unit1.Em6.ControlNodes".cm.softCam.mendrelAnodeFrontAxisZ.down.inPos )
   END_RUNG wire#w1
   RUNG wire#powerrail
      Contact( "Unit1.Em6.ControlNodes".cm.softCam.mendrelAnodeFrontAxisZ.up.inPos )
      Contact( "Unit1.Em6.ControlNodes".cm.softCam.mendrelAnodeFrontAxisY.backward.inPos )
   END_RUNG wire#w1
   RUNG wire#powerrail
      Contact( "Unit1.Em6.ControlNodes".cm.softCam.mendrelAnodeRearAxisZ.down.inPos )
   END_RUNG wire#w2
   RUNG wire#powerrail
      Contact( "Unit1.Em6.ControlNodes".cm.softCam.mendrelAnodeRearAxisZ.up.inPos )
      Contact( "Unit1.Em6.ControlNodes".cm.softCam.mendrelAnodeRearAxisY.backward.inPos )
   END_RUNG wire#w2
   RUNG wire#powerrail
      Contact( "Unit1.Em6.ControlNodes".cm.softCam.mendrelCathodeFrontAxisZ.down.inPos )
   END_RUNG wire#w3
   RUNG wire#powerrail
      Contact( "Unit1.Em6.ControlNodes".cm.softCam.mendrelCathodeFrontAxisZ.up.inPos )
      Contact( "Unit1.Em6.ControlNodes".cm.softCam.mendrelCathodeFrontAxisY.backward.inPos )
   END_RUNG wire#w3
   RUNG wire#powerrail
      Contact( "Unit1.Em6.ControlNodes".cm.softCam.mendrelCathodeRearAxisZ.down.inPos )
   END_RUNG wire#w4
   RUNG wire#powerrail
      Contact( "Unit1.Em6.ControlNodes".cm.softCam.mendrelCathodeRearAxisZ.up.inPos )
      Contact( "Unit1.Em6.ControlNodes".cm.softCam.mendrelCathodeRearAxisY.backward.inPos )
   END_RUNG wire#w4
   RUNG wire#powerrail
      I_Contact( #FALSE )
      I_Contact( "Unit1.Em6.ControlNodes".stackTable."step".action1[183] )
      Not()
      wire#w5
      Contact( "Unit1.Em6.ControlNodes".cm.Interlock.finalRollerFrontAxisX.source.posAbsolute[0] )
      Move(in := 0, out1 => "Unit1.Em6.ControlNodes".cmFinalRollerFrontAxisX.commands.selectSetPosition)
      Coil( "Unit1.Em6.ControlNodes".cm.Command.finalRollerFrontAxisX.posAbsolute[0] )
   END_RUNG
   RUNG wire#powerrail
      I_Contact( "Unit1.Em6.ControlNodes".gaugeRnR."step".action1[110] )
      Not()
   END_RUNG wire#w5
   // the same network as SCL:
   #instFinalRollerFrontAxisX_Position[0](PosiNo := 0,   // "Position.LER_Axis"
                           Status := #unitStatus,
                           int1 := "Unit1.Em6.ControlNodes".emRelations.em5.softCam.cathodeMainPnP2AxisX.alignTablePos.inPos,
                           int2 := "Unit1.Em6.ControlNodes".cm.softCam.mendrelAnodeFrontAxisZ.down.inPos OR ("Unit1.Em6.ControlNodes".cm.softCam.mendrelAnodeFrontAxisZ.up.inPos AND "Unit1.Em6.ControlNodes".cm.softCam.mendrelAnodeFrontAxisY.backward.inPos),
                           int3 := "Unit1.Em6.ControlNodes".cm.softCam.mendrelAnodeRearAxisZ.down.inPos OR ("Unit1.Em6.ControlNodes".cm.softCam.mendrelAnodeRearAxisZ.up.inPos AND "Unit1.Em6.ControlNodes".cm.softCam.mendrelAnodeRearAxisY.backward.inPos),
                           int4 := "Unit1.Em6.ControlNodes".cm.softCam.mendrelCathodeFrontAxisZ.down.inPos OR ("Unit1.Em6.ControlNodes".cm.softCam.mendrelCathodeFrontAxisZ.up.inPos AND "Unit1.Em6.ControlNodes".cm.softCam.mendrelCathodeFrontAxisY.backward.inPos),
                           int5 := "Unit1.Em6.ControlNodes".cm.softCam.mendrelCathodeRearAxisZ.down.inPos OR ("Unit1.Em6.ControlNodes".cm.softCam.mendrelCathodeRearAxisZ.up.inPos AND "Unit1.Em6.ControlNodes".cm.softCam.mendrelCathodeRearAxisY.backward.inPos),
                           commands := "Unit1.Em6.HmiInterface".cmFinalRollerFrontAxisX.commands,
                           interlockOk := "Unit1.Em6.ControlNodes".cm.Interlock.finalRollerFrontAxisX.source.posAbsolute,
                           intOut := "Unit1.Em6.HmiInterface".intCondition.Axis_21.Jog.intOut);
   #_w1 := (NOT (NOT #FALSE AND NOT "Unit1.Em6.ControlNodes".stackTable."step".action1[183]) OR NOT (NOT "Unit1.Em6.ControlNodes".gaugeRnR."step".action1[110])) AND "Unit1.Em6.ControlNodes".cm.Interlock.finalRollerFrontAxisX.source.posAbsolute[0];
   IF #_w1 THEN "Unit1.Em6.ControlNodes".cmFinalRollerFrontAxisX.commands.selectSetPosition := 0; END_IF;
   "Unit1.Em6.ControlNodes".cm.Command.finalRollerFrontAxisX.posAbsolute[0] := #_w1;
END_REGION

